// TwinCAT 3 PLC project SiftClient
// Title: Sift Client Library
// Company: Sift Stack Inc
// Author: Marc Julien
// ProjectVersion: 0.2.0.0
// Description: Sift Client library for streaming data from PLC applications into Sift.
// ProgramVersion: 3.1.4026.14
// libraries:
//   Tc2_Standard, * (Beckhoff Automation GmbH)
//   Tc2_System, * (Beckhoff Automation GmbH)
//   Tc2_TcpIp, * (Beckhoff Automation GmbH)
//   Tc2_Utilities, * (Beckhoff Automation GmbH)
//   Tc3_JsonXml, * (Beckhoff Automation GmbH)
//   TcUnit, * (www.tcunit.org)
// project tree:
//   DUTs/ E_ChannelDataType.TcDUT, ST_ChannelConfig.TcDUT, ST_EnumType.TcDUT, ST_FlowConfig.TcDUT, ST_IngestionConfig.TcDUT, T_SiftClient.TcDUT, ST_SiftError.TcDUT
//   DUTs/Private/ _ST_Timestamp.TcDUT, _ST_SiftMessage.TcDUT, _U_SiftChannelValue.TcDUT
//   GVLs/ GVL_SIFT.TcGVL, SiftClientParameters.TcGVL
//   / PlcTask.TcTTO
//   POUs/ FB_SiftClient.TcPOU
//   POUs/Private/ SAFE_MEMCPY.TcPOU, _FB_SendSiftMessage.TcPOU, _FB_BufferWriter.TcPOU, _F_CreateAuthenticateMessage.TcPOU, _F_CreateDataMessage.TcPOU, _F_CreateEndpointMessage.TcPOU, _F_CreateIngestionConfigMessage.TcPOU, _F_CreatePingMessage.TcPOU, _F_CreateRunMessage.TcPOU, _F_IsSuccessfulResponse.TcPOU, _F_SetSiftError.TcPOU
//   POUs/Services/ FB_IngestionConfigService.TcPOU, FB_IngestService.TcPOU, FB_PingService.TcPOU, FB_RunService.TcPOU
//   POUs/Services/Private/ FB_AuthenticateService.TcPOU
//   POUs/Util/ GetCurrentTime.TcPOU, SetChannelValue.TcPOU
//   Tests/ FB_BufferWriter_Test.TcPOU, FB_CreateDataMessage_Test.TcPOU, FB_CreateIngestionConfigMessage_Test.TcPOU, FB_CreatePingMessage_Test.TcPOU, FB_CreateRunMessage_Test.TcPOU, FB_SAFE_MEMCPY_Test.TcPOU, FB_SetChannelValue_Test.TcPOU, FB_SiftError_Test.TcPOU, PRG_TEST.TcPOU
//   Version/ Global_Version.TcGVL
// real-time tasks:
//   TASK PlcTask: cycle T#10ms, priority 20, ADS port 350

CONFIGURATION SiftClient
    RESOURCE PLC ON TwinCAT3
        TASK PlcTask(INTERVAL := T#10ms, PRIORITY := 20);
        PROGRAM PRG_TEST WITH PlcTask : PRG_TEST;
    END_RESOURCE
END_CONFIGURATION

// ---- DUTs/E_ChannelDataType.TcDUT
{attribute 'qualified_only'}
{attribute 'strict'}
{attribute 'to_string'}
TYPE E_ChannelDataType :
(
	Unspecified,
	Int32,
	Uint32,
	Int64,
	Uint64,
	Bool_,
	String_,
	Double,
	Float,
	Enum
);
END_TYPE

// ---- DUTs/Private/_ST_Timestamp.TcDUT
TYPE _ST_Timestamp :
STRUCT
	nSeconds : LINT;
	nNanoseconds : DINT;
END_STRUCT
END_TYPE

// ---- DUTs/Private/_ST_SiftMessage.TcDUT
TYPE _ST_SiftMessage :
STRUCT
	nType : BYTE;
	nLength : UDINT;
	aData : ARRAY[1..SiftClientParameters.MAX_PACKET_SIZE] OF BYTE;
END_STRUCT
END_TYPE

// ---- DUTs/Private/_U_SiftChannelValue.TcDUT
TYPE _U_SiftChannelValue :
UNION
	nInt32 : DINT;
	nUint32 : UDINT;
	nInt64 : LINT;
	nUint64 : ULINT;
	bBool : BOOL;
	fDouble : LREAL;
	fFloat : REAL;
	nEnum : UDINT;
	sString : STRING(255);
END_UNION
END_TYPE

// ---- DUTs/ST_ChannelConfig.TcDUT
TYPE ST_ChannelConfig :
STRUCT
	sName : STRING(255); 		   // This Channel's name. Required.
	eDataType : E_ChannelDataType; // This Channel's data type. Required.
	sDescription : STRING(255);	   // This Channel's description. Optional.
	sUnit : STRING(255);           // This Channel's units. Optional.
	// Enums for this channel. Required for Channels with the Enum data type.
	aEnumTypes : ARRAY[0..SiftClientParameters.MAX_NUM_ENUMS_PER_CHANNEL - 1] OF ST_EnumType;
	nNumEnumTypes : UDINT; // Total number of enums for this Channel.
	
	Value : _U_SiftChannelValue; // The current value of this Channel.
END_STRUCT
END_TYPE

// ---- DUTs/ST_EnumType.TcDUT
TYPE ST_EnumType :
STRUCT
	nKey : UDINT;        // Numerical key for this Enum.
	sName : STRING(255); // Name or label for this Enum.
END_STRUCT
END_TYPE

// ---- DUTs/ST_FlowConfig.TcDUT
TYPE ST_FlowConfig :
STRUCT
	sName : STRING(255); // This Flow's name.
	// The Channels in this Flow.
	aChannelConfigs : ARRAY[0..SiftClientParameters.MAX_NUM_CHANNELS_PER_FLOW - 1] OF ST_ChannelConfig;
	nNumChannelConfigs : UDINT; // Total number of channels in this Flow.
END_STRUCT
END_TYPE

// ---- DUTs/ST_IngestionConfig.TcDUT
TYPE ST_IngestionConfig :
STRUCT
	sAssetName : STRING(255); // Asset name for this Ingestion Config.
	// The Flows for this Ingestion Config.
	aFlowConfigs : ARRAY[0..SiftClientParameters.MAX_NUM_FLOWS - 1] OF ST_FlowConfig;
	nNumFlowConfigs : UDINT; // Total number of Flows in this Ingestion Config.
END_STRUCT
END_TYPE

// ---- DUTs/T_SiftClient.TcDUT
TYPE T_SiftClient :
STRUCT
	sHost : T_IPv4Addr; // Sift Proxy address.
	nPort : UINT;       // Sift Proxy port.
	
	sGrpcUri : STRING(255); // Sift gRPC URI.
	sApiKey : STRING;       // Sift API key.
	
	pJsonBuffer : POINTER TO BYTE; // Buffer used to create JSON messages.
	pJbLength : UDINT;			   // Size of pJsonBuffer.
	
   	fbCloseAll 		: FB_SocketCloseAll;
	fbConnect		: FB_SocketConnect;
	fbSend		    : FB_SocketSend;
	fbReceive     	: FB_SocketReceive;
	fbClose			: FB_SocketClose;
	
END_STRUCT
END_TYPE

// ---- DUTs/ST_SiftError.TcDUT
TYPE ST_SiftError :
STRUCT
	bError : BOOL;     // True is this is an error. 
	nErrId : UDINT;    // The ID of this error.
	sReason : STRING;  // Error message in string format.
END_STRUCT
END_TYPE

// ---- GVLs/GVL_SIFT.TcGVL
{attribute 'qualified_only'}
VAR_GLOBAL CONSTANT
	//Defaults
	SIFT_PROXY_CMD_ARGS : STRING(255) := '--stream_metrics --storage_path %s --listen_port=%d --grpc_uri=%s --api_key=%s tcp sift_proxy --little_endian --end_stream_on_error --verbose';
	SIFT_PROXY_DEFAULT_HOST : T_IPv4Addr := '127.0.0.1';
	SIFT_PROXY_DEFAULT_LISTEN_PORT : UINT := 10010;
	SIFT_PROXY_START_DELAY : TIME := T#5S;
	
	SYNC_WORD : UDINT := 16#ABCDEF00;
	HEADER_LENGTH : UDINT := 9;
	MESSAGE_TYPE_INDEX : BYTE := 4;
	MESSGE_LENGTH_INDEX : BYTE := 5;

	ENDPOINT_MESSAGE_TYPE : BYTE := 16#01;
	DATA_MESSAGE_TYPE : BYTE := 16#02;
	RESPONSE_MESSAGE_TYPE : BYTE := 16#FF;
	
	SIFT_CLIENT_DEFAULT_LOCAL_IP : T_IPv4Addr := '127.0.0.1';
	SIFT_CLIENT_DEFAULT_LOCAL_PORT : UINT := 10009;
	
	MAX_JSON_RESPONSE_SIZE : UDINT := 1024; // Max JSON response size.
		
	(* Error Codes *)
	BUFFER_CAPACITY_REACHED : UDINT := 16#5000_0000; // Buffer is at capacity.
	JSON_CAPACITY_REACHED : UDINT := 16#5000_0001; // JSON message is too large. Should increase JSON buffer size.
	NULL_JSON_POINTER : UDINT := 16#5000_0002; // The JSON buffer passed in is Null.
	INGEST_RING_BUFFER_REMOVE_ERROR : UDINT := 16#5000_0003; // Error removing data from ingest ring buffer.
	MEMCPY_ERROR : UDINT := 16#5000_0004; // Error calling MEMCPY
	BAD_PARAMETERS : UDINT := 16#5000_0005; // User has configured the parameters incorrectly.
	UNABLE_TO_PARSE_JSON : UDINT := 16#5000_0005; // Internal JSON could not be parsed.
	
	SIFT_PROXY_NO_RESPONSE : UDINT := 16#5000_1000; // No response from Sift Proxy
	SIFT_PROXY_FAILED_TO_START : UDINT := 16#5000_1001;  // Failed to start Sift Proxy
	SIFT_PROXY_INVALID_RESPONSE : UDINT := 16#5000_1002;  // Invalid response from Sift Proxy
	SIFT_PROXY_INVALID_SYNC_WORD : UDINT := 16#5000_1003;  // Invalid sync word from Sift Proxy
	SIFT_PROXY_SIFT_API_ERROR : UDINT := 16#5000_1004;  // Invalid argument to the endpoint
	
	INVALID_GRPC_URI : UDINT := 16#5000_2000;
	INVALID_API_KEY : UDINT := 16#5000_2001;
	INVALID_INGESTION_CONFIG : UDINT := 16#5000_2002;
    INVALID_LOG_DIR : UDINT := 16#5000_2003;
	
END_VAR

// ---- GVLs/SiftClientParameters.TcGVL
{attribute 'qualified_only'}
VAR_GLOBAL CONSTANT
	// The path to the `start_sift_proxy.bat` file.
	START_SIFT_PROXY_PATH : STRING := 'C:\Sift\Beckhoff\start_sift_proxy.bat';
		
	MAX_NUM_FLOWS : UDINT := 8; // Max number of Flows per Ingestion Config.
	MAX_NUM_CHANNELS_PER_FLOW : UDINT := 256; // Max number of Channels per Flow.
	MAX_NUM_ENUMS_PER_CHANNEL : UDINT := 256; // Max number of Enums per Channel.
	MAX_NUM_TAGS : UDINT := 32; // Max number of tags (for a run).
	
	// Maximum size of a single Sift packet. 
	// This should be large enough to fit all configured flows at once
	// and also large enough to fit the ingestion config request.
	MAX_PACKET_SIZE : UDINT := 8192;
	
END_VAR

// ---- Version/Global_Version.TcGVL
{attribute 'TcGenerated'}
{attribute 'no-analysis'}
{attribute 'linkalways'}
// This function has been automatically generated from the project information.
VAR_GLOBAL CONSTANT
	{attribute 'const_non_replaced'}
	stLibVersion_Sift_Client_Library : ST_LibVersion := (iMajor := 0, iMinor := 1, iBuild := 0, iRevision := 0, nFlags := 0, sVersion := '0.1.0.0');
END_VAR

// ---- Tests/PRG_TEST.TcPOU
PROGRAM PRG_TEST
VAR
	fbSetChannelValue_Test : FB_SetChannelValue_Test;
	fbSafeMemcpy_Test : FB_SAFE_MEMCPY_Test;
	fbBufferWriter_Test : FB_BufferWriter_Test;
	fbCreateIngestionConfigMessage_Test: FB_CreateIngestionConfigMessage_Test;
	fbCreatePingMessage_Test : FB_CreatePingMessage_Test;
	fbCreateRunMessage_Test : FB_CreateRunMessage_Test;
	fbSiftError_Test : FB_SiftError_Test;
	fbCreateDataMessage_Test : FB_CreateDataMessage_Test;
END_VAR

TcUnit.RUN();

END_PROGRAM

// ---- Tests/FB_SetChannelValue_Test.TcPOU
FUNCTION_BLOCK FB_SetChannelValue_Test EXTENDS TcUnit.FB_TestSuite
VAR_INPUT
END_VAR

VAR_OUTPUT
END_VAR

VAR
	stIngestionConfig : ST_IngestionConfig;
	fbIngestionConfig : FB_IngestionConfigService := (stIngestionConfig := stIngestionConfig);
	pFlowConfig : POINTER TO ST_FlowConfig;
	pChannel : POINTER TO ST_ChannelConfig;
END_VAR

Nominal();
Invalid();

METHOD Invalid : REFERENCE TO FB_Test
VAR_INPUT
	bBoolTestValue : BOOL := TRUE;
	fDoubleTestValue : LREAL := 1.2345;
	nEnumTestValue : UDINT := 10;
	fFloatTestValue : REAL := 9.8765;
	nInt32TestValue : DINT := 12345;
	sStringTestValue : STRING(255) := 'Test string value';
	nUInt32TestValue : UDINT := 4893573;
	nInt64TestValue : LINT := -12232423;
	nUInt64TestValue : ULINT := 1249864785;
END_VAR
TEST('SetChannelValue Invalid');

pFlowConfig := fbIngestionConfig.CreateFlowConfig('flow_name');

// Null
AssertFalse(SetChannelValue(pChannel := pChannel, fDoubleTestValue),
            Message := 'setting a null pointer should have failed');

// BOOL
pChannel := fbIngestionConfig.CreateChannelConfig(pFlowConfig := pFlowConfig,
                                                  sName := 'bool_channel',
                                                  E_ChannelDataType.Bool_,
                                                  sDescription := '',
                                                  sUnit := '');				  
AssertFalse(SetChannelValue(pChannel := pChannel, fDoubleTestValue),
            Message := 'setting the bool value should have failed');

// STRING
pChannel := fbIngestionConfig.CreateChannelConfig(pFlowConfig := pFlowConfig,
                                                  sName := 'string_channel',
                                                  E_ChannelDataType.String_,
                                                  sDescription := '',
                                                  sUnit := '');
AssertFalse(SetChannelValue(pChannel := pChannel, nUInt32TestValue),
            Message := 'setting the string value should have failed');

// DOUBLE
pChannel := fbIngestionConfig.CreateChannelConfig(pFlowConfig := pFlowConfig,
                                                  sName := 'double_channel',
                                                  E_ChannelDataType.Double,
                                                  sDescription := '',
                                                  sUnit := '');				  
AssertFalse(SetChannelValue(pChannel := pChannel, nEnumTestValue),
            Message := 'setting the string value should have failed');

// FLOAT
pChannel := fbIngestionConfig.CreateChannelConfig(pFlowConfig := pFlowConfig,
                                                  sName := 'float_channel',
                                                  E_ChannelDataType.Float,
                                                  sDescription := '',
                                                  sUnit := '');				  
AssertFalse(SetChannelValue(pChannel := pChannel, nInt32TestValue),
            Message := 'setting the float value should have failed');

// ENUM
pChannel := fbIngestionConfig.CreateChannelConfig(pFlowConfig := pFlowConfig,
                                                  sName := 'enum_channel',
                                                  E_ChannelDataType.Enum,
                                                  sDescription := '',
                                                  sUnit := '');				  
AssertFalse(SetChannelValue(pChannel := pChannel, fFloatTestValue),
            Message := 'setting the enum value should have failed');

// INT32
pChannel := fbIngestionConfig.CreateChannelConfig(pFlowConfig := pFlowConfig,
                                                  sName := 'int32_channel',
                                                  E_ChannelDataType.Int32,
                                                  sDescription := '',
                                                  sUnit := '');				  
AssertFalse(SetChannelValue(pChannel := pChannel, sStringTestValue),
            Message := 'setting the int32 value should have failed');

// UINT32
pChannel := fbIngestionConfig.CreateChannelConfig(pFlowConfig := pFlowConfig,
                                                  sName := 'uint32_channel',
                                                  E_ChannelDataType.Uint32,
                                                  sDescription := '',
                                                  sUnit := '');				  
AssertFalse(SetChannelValue(pChannel := pChannel, nInt64TestValue),
            Message := 'setting the uint32 value should have failed');

// INT64
pChannel := fbIngestionConfig.CreateChannelConfig(pFlowConfig := pFlowConfig,
                                                  sName := 'int64_channel',
                                                  E_ChannelDataType.Int64,
                                                  sDescription := '',
                                                  sUnit := '');				  
AssertFalse(SetChannelValue(pChannel := pChannel, nUInt64TestValue),
            Message := 'setting the int64 value should have failed');

// UINT64
pChannel := fbIngestionConfig.CreateChannelConfig(pFlowConfig := pFlowConfig,
                                                  sName := 'uint64_channel',
                                                  E_ChannelDataType.Uint64,
                                                  sDescription := '',
                                                  sUnit := '');				  
AssertFalse(SetChannelValue(pChannel := pChannel, bBoolTestValue),
            Message := 'setting the uint64 value should have failed');


TEST_FINISHED();
END_METHOD

METHOD Nominal : REFERENCE TO FB_Test
VAR_INPUT
END_VAR

VAR
	bBoolTestValue : BOOL := TRUE;
	fDoubleTestValue : LREAL := 1.2345;
	nEnumTestValue : UDINT := 10;
	fFloatTestValue : REAL := 9.8765;
	nInt32TestValue : DINT := 12345;
	sStringTestValue : STRING(255) := 'Test string value';
	nUInt32TestValue : UDINT := 4893573;
	nInt64TestValue : LINT := -12232423;
	nUInt64TestValue : ULINT := 1249864785;
END_VAR
TEST('SetChannelValue Nominal');

pFlowConfig := fbIngestionConfig.CreateFlowConfig('flow_name');

// BOOL
pChannel := fbIngestionConfig.CreateChannelConfig(pFlowConfig := pFlowConfig,
                                                  sName := 'bool_channel',
                                                  E_ChannelDataType.Bool_,
                                                  sDescription := '',
                                                  sUnit := '');				  
AssertTrue(SetChannelValue(pChannel := pChannel, bBoolTestValue),
           Message := 'the bool value was not set correctly');
AssertEquals_BOOL(Expected := bBoolTestValue, 
                  Actual := pChannel^.Value.bBool,
                  Message := 'the bool value is incorrect');

// STRING
pChannel := fbIngestionConfig.CreateChannelConfig(pFlowConfig := pFlowConfig,
                                                  sName := 'string_channel',
                                                  E_ChannelDataType.String_,
                                                  sDescription := '',
                                                  sUnit := '');
AssertTrue(SetChannelValue(pChannel := pChannel, sStringTestValue),
           Message := 'the string value was not set correctly');
AssertEquals_STRING(Expected := sStringTestValue, 
                    Actual := pChannel^.Value.sString,
                    Message := 'the string value is incorrect');

// DOUBLE
pChannel := fbIngestionConfig.CreateChannelConfig(pFlowConfig := pFlowConfig,
                                                  sName := 'double_channel',
                                                  E_ChannelDataType.Double,
                                                  sDescription := '',
                                                  sUnit := '');				  
AssertTrue(SetChannelValue(pChannel := pChannel, fDoubleTestValue),
           Message := 'the double value was not set correctly');
AssertEquals_LREAL(Expected := fDoubleTestValue, 
                   Actual := pChannel^.Value.fDouble,
                   Message := 'the double value is incorrect',
                   Delta := 0.0);

// FLOAT
pChannel := fbIngestionConfig.CreateChannelConfig(pFlowConfig := pFlowConfig,
                                                  sName := 'float_channel',
                                                  E_ChannelDataType.Float,
                                                  sDescription := '',
                                                  sUnit := '');				  
AssertTrue(SetChannelValue(pChannel := pChannel, fFloatTestValue),
           Message := 'the float value was not set correctly');
AssertEquals_REAL(Expected := fFloatTestValue, 
                  Actual := pChannel^.Value.fFloat,
                  Message := 'the float value is incorrect',
                  Delta := 0.0);

// ENUM
pChannel := fbIngestionConfig.CreateChannelConfig(pFlowConfig := pFlowConfig,
                                                  sName := 'enum_channel',
                                                  E_ChannelDataType.Enum,
                                                  sDescription := '',
                                                  sUnit := '');				  
AssertTrue(SetChannelValue(pChannel := pChannel, nEnumTestValue),
           Message := 'the enum value was not set correctly');
AssertEquals_UDINT(Expected := nEnumTestValue, 
                   Actual := pChannel^.Value.nEnum,
                   Message := 'the enum value is incorrect');

// INT32
pChannel := fbIngestionConfig.CreateChannelConfig(pFlowConfig := pFlowConfig,
                                                  sName := 'int32_channel',
                                                  E_ChannelDataType.Int32,
                                                  sDescription := '',
                                                  sUnit := '');				  
AssertTrue(SetChannelValue(pChannel := pChannel, nInt32TestValue),
           Message := 'the int32 value was not set correctly');
AssertEquals_DINT(Expected := nInt32TestValue, 
                  Actual := pChannel^.Value.nInt32,
                  Message := 'the int32 value is incorrect');

// UINT32
pChannel := fbIngestionConfig.CreateChannelConfig(pFlowConfig := pFlowConfig,
                                                  sName := 'uint32_channel',
                                                  E_ChannelDataType.Uint32,
                                                  sDescription := '',
                                                  sUnit := '');				  
AssertTrue(SetChannelValue(pChannel := pChannel, nUInt32TestValue),
           Message := 'the uint32 value was not set correctly');
AssertEquals_UDINT(Expected := nUInt32TestValue, 
                   Actual := pChannel^.Value.nUInt32,
                   Message := 'the uint32 value is incorrect');

// INT64
pChannel := fbIngestionConfig.CreateChannelConfig(pFlowConfig := pFlowConfig,
                                                  sName := 'int64_channel',
                                                  E_ChannelDataType.Int64,
                                                  sDescription := '',
                                                  sUnit := '');				  
AssertTrue(SetChannelValue(pChannel := pChannel, nInt64TestValue),
           Message := 'the int64 value was not set correctly');
AssertEquals_LINT(Expected := nInt64TestValue, 
                  Actual := pChannel^.Value.nInt64,
                  Message := 'the int64 value is incorrect');

// UINT64
pChannel := fbIngestionConfig.CreateChannelConfig(pFlowConfig := pFlowConfig,
                                                  sName := 'uint64_channel',
                                                  E_ChannelDataType.Uint64,
                                                  sDescription := '',
                                                  sUnit := '');				  
AssertTrue(SetChannelValue(pChannel := pChannel, nUInt64TestValue),
           Message := 'the uint64 value was not set correctly');
AssertEquals_ULINT(Expected := nUInt64TestValue, 
                   Actual := pChannel^.Value.nUInt64,
                   Message := 'the uint64 value is incorrect');

TEST_FINISHED();
END_METHOD

END_FUNCTION_BLOCK

// ---- POUs/Services/FB_IngestionConfigService.TcPOU
// Service for creating and sending an Ingestion Config.
// The Ingestion Config is sent on the rising edge of bExecute.
FUNCTION_BLOCK FB_IngestionConfigService
VAR_INPUT
	hSiftClient : REFERENCE TO T_SiftClient;
	sAssetName : STRING(255);
	bExecute : BOOL;
	
END_VAR
VAR_OUTPUT
	bBusy : BOOL;
	bError : BOOL;
	nErrId : UDINT;
	sId : STRING(255);
	stIngestionConfig : ST_IngestionConfig;
	stSiftError : ST_SiftError;
END_VAR
VAR
	eState : (IDLE, SEND_MESSAGE, WAIT_FOR_RESPONSE, SUCCESS, FAILURE) := IDLE;
	fbSendSiftMessage : _FB_SendSiftMessage;
	stConfigReq : _ST_SiftMessage;
	fbJson : FB_JsonDomParser;
	sResponse : STRING(GVL_SIFT.MAX_JSON_RESPONSE_SIZE);
	jsonDoc : SJsonValue;
END_VAR

stIngestionConfig.sAssetName := sAssetName;
		
CASE eState OF
	IDLE:		
		IF bExecute THEN
			eState := SEND_MESSAGE;
		END_IF
		
	SEND_MESSAGE:
		bBusy := TRUE;
		bError := FALSE;
		stSiftError := _F_CreateIngestionConfigMessage(stIngestionConfig := stIngestionConfig, 
													   stMsg := stConfigReq,
													   pJsonBuffer := hSiftClient.pJsonBuffer,
													   nLength := hSiftClient.pJbLength);
		IF stSiftError.bError THEN
			nErrId := stSiftError.nErrId;
			eState := FAILURE;
			RETURN;
		END_IF
		fbSendSiftMessage(hSiftClient := hSiftClient, stMsg := stConfigReq, bExecute := TRUE);
		eState := WAIT_FOR_RESPONSE;

	WAIT_FOR_RESPONSE:
		bBusy := TRUE;
		bError := FALSE;
		fbSendSiftMessage(bExecute := FALSE);
		
		IF fbSendSiftMessage.bBusy THEN
			RETURN;
		ELSIF fbSendSiftMessage.bError THEN
			nErrId := fbSendSiftMessage.nErrId;
			eState := FAILURE;
			RETURN;
		END_IF
		
		// Verify response.
		IF fbSendSiftMessage.stResponse.nLength > GVL_SIFT.MAX_JSON_RESPONSE_SIZE THEN
			nErrId := GVL_SIFT.JSON_CAPACITY_REACHED;
			eState := FAILURE;
			RETURN;	
		END_IF
		
		IF NOT SAFE_MEMCPY(ADR(sResponse), SIZEOF(sResponse), 
			               ADR(fbSendSiftMessage.stResponse.aData), fbSendSiftMessage.stResponse.nLength) THEN
			nErrId := GVL_SIFT.MEMCPY_ERROR;
			eState := FAILURE;
		END_IF
		
		jsonDoc := fbJson.ParseDocument(sResponse);
		IF jsonDoc = 0 THEN
			eState := FAILURE;
			nErrId := GVL_SIFT.UNABLE_TO_PARSE_JSON;
		END_IF
		
		IF _F_IsSuccessfulResponse(jsonDoc) THEN
			IF NOT fbJson.HasMember(jsonDoc, 'data') THEN
				nErrId := GVL_SIFT.SIFT_PROXY_INVALID_RESPONSE;
				eState := FAILURE;
				RETURN;
			END_IF
			
			jsonDoc := fbJson.FindMember(jsonDoc, 'data');	
			IF NOT fbJson.HasMember(jsonDoc, 'ingestionConfig') THEN
				nErrId := GVL_SIFT.SIFT_PROXY_INVALID_RESPONSE;
				eState := FAILURE;
				RETURN;
			END_IF

			jsonDoc := fbJson.FindMember(jsonDoc, 'ingestionConfig');
			IF NOT fbJson.HasMember(jsonDoc, 'ingestionConfigId') THEN
				nErrId := GVL_SIFT.SIFT_PROXY_INVALID_RESPONSE;
				eState := FAILURE;
				RETURN;
			END_IF
			
			jsonDoc := fbJson.FindMember(jsonDoc, 'ingestionConfigId');
			sId := fbJson.GetString(jsonDoc);
			
			eState := SUCCESS;
		ELSE
			IF NOT _F_SetSiftError(jsonDoc, stSiftError) THEN
				nErrId := GVL_SIFT.SIFT_PROXY_INVALID_RESPONSE;
				RETURN;
			END_IF
			nErrId := stSiftError.nErrId;
			eState := FAILURE;
		END_IF
		
	SUCCESS:
		bBusy := FALSE;
		bError := FALSE;
		eState := IDLE;
		
	FAILURE:
		bBusy := FALSE;
		bError := TRUE;
		eState := IDLE;
END_CASE

METHOD ClearIngestionConfig : BOOL
VAR_INPUT
END_VAR

VAR
	i,j : UDINT;
END_VAR
FOR i := 1 TO stIngestionConfig.nNumFlowConfigs DO
	FOR j := 1 TO stIngestionConfig.aFlowConfigs[i-1].nNumChannelConfigs DO
    	stIngestionConfig.aFlowConfigs[i-1].aChannelConfigs[j-1].sName := '';
		stIngestionConfig.aFlowConfigs[i-1].aChannelConfigs[j-1].sDescription := '';
		stIngestionConfig.aFlowConfigs[i-1].aChannelConfigs[j-1].sUnit := '';
		stIngestionConfig.aFlowConfigs[i-1].aChannelConfigs[j-1].eDataType := E_ChannelDataType.Unspecified;
		stIngestionConfig.aFlowConfigs[i-1].aChannelConfigs[j-1].nNumEnumTypes := 0;
	END_FOR
	stIngestionConfig.aFlowConfigs[i-1].nNumChannelConfigs := 0;
	stIngestionConfig.aFlowConfigs[i-1].sName := '';
END_FOR
stIngestionConfig.sAssetName := '';
stIngestionConfig.nNumFlowConfigs := 0;
END_METHOD

METHOD CreateChannelConfig : POINTER TO ST_ChannelConfig
VAR_INPUT
	pFlowConfig : POINTER TO ST_FlowConfig;
	sName : STRING(255);
	eDataType : E_ChannelDataType;
	sDescription : STRING(255);
	sUnit : STRING(255);
END_VAR
VAR 
	pChannelConfig : POINTER TO ST_ChannelConfig;
END_VAR
IF pFlowConfig = 0 THEN
	CreateChannelConfig := 0;
	RETURN;
END_IF

IF pFlowConfig^.nNumChannelConfigs >= SiftClientParameters.MAX_NUM_CHANNELS_PER_FLOW THEN
	CreateChannelConfig := 0;
	RETURN;
END_IF

pChannelConfig := ADR(pFlowConfig^.aChannelConfigs[pFlowConfig^.nNumChannelConfigs]);
pChannelConfig^.sName := sName;
pChannelConfig^.eDataType := eDataType;
pChannelConfig^.sDescription := sDescription;
pChannelConfig^.sUnit := sUnit;

pFlowConfig^.nNumChannelConfigs := pFlowConfig^.nNumChannelConfigs + 1;
CreateChannelConfig := pChannelConfig;
END_METHOD

METHOD CreateFlowConfig : POINTER TO ST_FlowConfig
VAR_INPUT
	sName : STRING(255);
END_VAR
IF stIngestionConfig.nNumFlowConfigs >= SiftClientParameters.MAX_NUM_FLOWS THEN
	CreateFlowConfig := 0;
	RETURN;
END_IF

stIngestionConfig.aFlowConfigs[stIngestionConfig.nNumFlowConfigs].sName := sName;
CreateFlowConfig := ADR(stIngestionConfig.aFlowConfigs[stIngestionConfig.nNumFlowConfigs]);

stIngestionConfig.nNumFlowConfigs := stIngestionConfig.nNumFlowConfigs + 1;
END_METHOD

METHOD InitEnumTypes : BOOL
VAR_INPUT
	pChannelConfig : POINTER TO ST_ChannelConfig;
	aEnumTypes : REFERENCE TO ARRAY[0..SiftClientParameters.MAX_NUM_ENUMS_PER_CHANNEL - 1] OF ST_EnumType;
END_VAR

VAR 
	i : UDINT;
END_VAR
IF pChannelConfig = 0 THEN
	InitEnumTypes := FALSE;
	RETURN;
END_IF

IF pChannelConfig^.eDataType <> E_ChannelDataType.Enum THEN
	InitEnumTypes := FALSE;
	RETURN;
END_IF


FOR i := 1 TO SiftClientParameters.MAX_NUM_ENUMS_PER_CHANNEL DO
	IF aEnumTypes[i-1].sName = '' THEN
		CONTINUE;
	END_IF
	
	pChannelConfig^.aEnumTypes[i-1] := aEnumTypes[i-1];
	pChannelConfig^.nNumEnumTypes := pChannelConfig^.nNumEnumTypes + 1;
END_FOR

InitEnumTypes := TRUE;
END_METHOD

// Resets the Ingestion Config service.
METHOD PUBLIC Reset : BOOL
VAR_INPUT
END_VAR
Reset := ClearIngestionConfig();
END_METHOD

METHOD PUBLIC Validate : BOOL
VAR_INPUT
END_VAR
VAR
	nSizeInBytes : UDINT;
	i : UDINT;
	j : UDINT;
	tmpChannelConfig : REFERENCE TO ST_ChannelConfig;
END_VAR
FOR i := 1 TO stIngestionConfig.nNumFlowConfigs DO
	FOR j := 1 TO stIngestionConfig.aFlowConfigs[i-1].nNumChannelConfigs DO
		tmpChannelConfig REF= stIngestionConfig.aFlowConfigs[i-1].aChannelConfigs[j-1];

		CASE tmpChannelConfig.eDataType OF
			E_ChannelDataType.Bool_:
				nSizeInBytes := nSizeInBytes + 1;
			
			E_ChannelDataType.Double:
				nSizeInBytes := nSizeInBytes + 8;
			
			E_ChannelDataType.Enum:
				nSizeInBytes := nSizeInBytes + 4;
			
			E_ChannelDataType.Float:
				nSizeInBytes := nSizeInBytes + 4;
			
			E_ChannelDataType.Int32:
				nSizeInBytes := nSizeInBytes + 4;
			
			E_ChannelDataType.Int64:
				nSizeInBytes := nSizeInBytes + 8;
			
			E_ChannelDataType.String_:
				nSizeInBytes := nSizeInBytes + 255;
			
			E_ChannelDataType.Uint32:
				nSizeInBytes := nSizeInBytes + 4;

			E_ChannelDataType.Uint64:
				nSizeInBytes := nSizeInBytes + 8;
		END_CASE
		
		IF tmpChannelConfig.eDataType = E_ChannelDataType.Unspecified THEN
			Validate := FALSE;
			RETURN;
		END_IF
	END_FOR
END_FOR

Validate := nSizeInBytes < SiftClientParameters.MAX_PACKET_SIZE;
END_METHOD

END_FUNCTION_BLOCK

// ---- POUs/Private/_FB_SendSiftMessage.TcPOU
// Sends a message to Sift Proxy using the Sift Proxy Protocol and waits for a response.
FUNCTION_BLOCK _FB_SendSiftMessage
VAR_INPUT
	hSiftClient : REFERENCE TO T_SiftClient;
	stMsg : REFERENCE TO _ST_SiftMessage;
	bExecute : BOOL;
	bWaitForReply : BOOL := TRUE;
	tReplyTimeout : TIME := T#10S; // Default 10s timeout. In practice we've seen local repsonses take up to about 1s.
END_VAR
VAR_OUTPUT
	bBusy : BOOL;
	bError : BOOL;
	stResponse : _ST_SiftMessage;
	nErrId : UDINT;
END_VAR

VAR
	eState : (IDLE, SEND_MESSAGE, SEND_MESSAGE_WAIT, RECEIVE_REPLY_START_TIMER, RECEIVE_REPLY, RECEIVE_REPLY_WAIT, SUCCESS, FAILURE):= IDLE;
	aRawBuf : ARRAY[1..SiftClientParameters.MAX_PACKET_SIZE] OF BYTE; // For the BufferWriter. Used for sending/receiving.
	fbWriter : _FB_BufferWriter := (pRawBuf := ADR(aRawBuf), nSize := SIZEOF(aRawBuf));	
	aRecvBuf : ARRAY[1..SiftClientParameters.MAX_PACKET_SIZE] OF BYTE; // Used for immediate recv calls.
	responseTimer : TON; // Timer for how longer to wait for a response from sift_proxy.
	nBytesRead : UDINT; // Current offset into the recv message.
	nRecvSyncWord : UDINT;	
	nRecvCount : UDINT;
END_VAR

CASE eState OF
	IDLE:
		IF bExecute THEN
			eState := SEND_MESSAGE;
		END_IF
		
	SEND_MESSAGE:
		bBusy := TRUE;
		bError := FALSE;
		
		// Always reset the writer before using it.
		fbWriter.SetOffset(0);
		
		// Verify MAX_PACKET_SIZE is a reasonable number
		IF SiftClientParameters.MAX_PACKET_SIZE <= GVL_SIFT.HEADER_LENGTH THEN
			nErrId := GVL_SIFT.BAD_PARAMETERS;
			eState := FAILURE;
			RETURN;
		END_IF
		
		// Sync word
		IF NOT fbWriter.Write(ADR(GVL_SIFT.SYNC_WORD), 4) THEN
			nErrId := GVL_SIFT.MEMCPY_ERROR;
			eState := FAILURE;
			RETURN;
		END_IF
		
		// Message type		
		IF NOT fbWriter.Write(ADR(stMsg.nType), 1) THEN
			nErrId := GVL_SIFT.MEMCPY_ERROR;
			eState := FAILURE;
			RETURN;
		END_IF
		
		// Message length
		IF NOT fbWriter.Write(ADR(stMsg.nLength), 4) THEN
			nErrId := GVL_SIFT.MEMCPY_ERROR;
			eState := FAILURE;
			RETURN;
		END_IF
			
		// Data.
		IF NOT fbWriter.Write(ADR(stMsg.aData), stMsg.nLength) THEN
			nErrId := GVL_SIFT.MEMCPY_ERROR;
			eState := FAILURE;
			RETURN;
		END_IF
		
		hSiftClient.fbSend(
			hSocket := hSiftClient.fbConnect.hSocket, 
			pSrc := ADR(aRawBuf),
			cbLen := stMsg.nLength + GVL_SIFT.HEADER_LENGTH,
			bExecute := TRUE,
		);
	
		eState := SEND_MESSAGE_WAIT;

	SEND_MESSAGE_WAIT:
		bBusy := TRUE;
		bError := FALSE;
		hSiftClient.fbSend(bExecute := FALSE);
		
		IF hSiftClient.fbSend.bBusy THEN
			RETURN;
		ELSIF hSiftClient.fbSend.bError THEN
			nErrId := hSiftClient.fbSend.nErrId;
			eState := FAILURE;
			RETURN;
		END_IF
		
		IF bWaitForReply THEN
			eState := RECEIVE_REPLY_START_TIMER;
		ELSE
			eState := SUCCESS;
		END_IF
	
	RECEIVE_REPLY_START_TIMER:
		bBusy := TRUE;
		bError := FALSE;
		responseTimer(IN:=FALSE);
		responseTimer(IN:=TRUE, PT:=tReplyTimeout);
		eState := RECEIVE_REPLY;
		nBytesRead := 0;
		
	RECEIVE_REPLY:
		bBusy := TRUE;
		bError := FALSE;

		hSiftClient.fbReceive(
			hSocket := hSiftClient.fbConnect.hSocket,
			cbLen := SiftClientParameters.MAX_PACKET_SIZE,
			pDest := ADR(aRecvBuf),
			bExecute := TRUE,
		);
		eState := RECEIVE_REPLY_WAIT;
		
	RECEIVE_REPLY_WAIT:
		bBusy := TRUE;
		bError := FALSE;
		hSiftClient.fbReceive(bExecute := FALSE);
		responseTimer();
				
		IF hSiftClient.fbReceive.bBusy THEN
			RETURN;
		ELSIF hSiftClient.fbReceive.bError THEN
			IF responseTimer.Q THEN
				nErrId := hSiftClient.fbReceive.nErrId;
				eState := FAILURE;
			ELSE
				eState := RECEIVE_REPLY;
			END_IF
			RETURN;
		END_IF
		
		IF hSiftClient.fbReceive.nRecBytes = 0 THEN
			IF responseTimer.Q THEN
				eState := FAILURE;
				nErrId := GVL_SIFT.SIFT_PROXY_NO_RESPONSE;
			ELSE	
				eState := RECEIVE_REPLY;
			END_IF		
			RETURN;
		END_IF
		
		// Always reset the writer before using it.
		fbWriter.SetOffset(0);
			
		IF NOT fbWriter.Write(ADR(aRecvBuf), hSiftClient.fbReceive.nRecBytes) THEN
			nErrId := GVL_SIFT.MEMCPY_ERROR;
			eState := FAILURE;
			RETURN;
		END_IF
		
		// If we have a complete header.
		IF fbWriter.nCurOffset >= GVL_SIFT.HEADER_LENGTH THEN
			IF NOT SAFE_MEMCPY(ADR(nRecvSyncWord), SIZEOF(nRecvSyncWord), ADR(aRawBuf), 4) THEN
				nErrId := GVL_SIFT.MEMCPY_ERROR;
				eState := FAILURE;
				RETURN;
			END_IF
			IF nRecvSyncWord <> GVL_SIFT.SYNC_WORD THEN
				eState := FAILURE;
				nErrId := GVL_SIFT.SIFT_PROXY_INVALID_SYNC_WORD;;
				RETURN;
			END_IF
			
			stResponse.nType := aRawBuf[GVL_SIFT.MESSAGE_TYPE_INDEX+1];
			IF stResponse.nType <> GVL_SIFT.RESPONSE_MESSAGE_TYPE THEN
				eState := FAILURE;
				nErrId := GVL_SIFT.SIFT_PROXY_INVALID_RESPONSE;;
				RETURN;
			END_IF	
			
			IF NOT SAFE_MEMCPY(ADR(stResponse.nLength), SIZEOF(stResponse.nLength), ADR(aRawBuf[GVL_SIFT.MESSGE_LENGTH_INDEX+1]), 4) THEN
				nErrId := GVL_SIFT.MEMCPY_ERROR;
				eState := FAILURE;
				RETURN;
			END_IF

			// Verify that the size of this message isn't larger than our buffer.
			IF stResponse.nLength > SIZEOF(stResponse.aData) THEN
				eState := FAILURE;
				nErrId := GVL_SIFT.BUFFER_CAPACITY_REACHED;
				RETURN;
			END_IF
			
			// Check if we have the whole packet
			IF fbWriter.nCurOffset >= GVL_SIFT.HEADER_LENGTH + stResponse.nLength THEN
				IF NOT SAFE_MEMCPY(ADR(stResponse.aData), SIZEOF(stResponse.aData),
								   ADR(aRawBuf[GVL_SIFT.HEADER_LENGTH+1]), stResponse.nLength) THEN
					nErrId := GVL_SIFT.MEMCPY_ERROR;
					eState := FAILURE;
					RETURN;
				END_IF
				
			ELSE // Incomplete packet.
				eState := RECEIVE_REPLY;
				RETURN;
			END_IF

		ELSE // Incomplete header.
			eState := RECEIVE_REPLY;
			RETURN;
		END_IF
		
		eState := SUCCESS;
		
	SUCCESS:
		bBusy := FALSE;
		bError := FALSE;
		eState := IDLE;
		
	FAILURE:
		bBusy := FALSE;
		bError := TRUE;
		eState := IDLE;
END_CASE

END_FUNCTION_BLOCK

// ---- POUs/Private/_FB_BufferWriter.TcPOU
// Helper for writing bytes to an array buffer.
FUNCTION_BLOCK _FB_BufferWriter
VAR_INPUT
	pRawBuf : POINTER TO BYTE; 
	nSize : UDINT;
END_VAR

VAR_OUTPUT
	nCurOffset : UDINT;
END_VAR

VAR
END_VAR

METHOD SetOffset : BOOL
VAR_INPUT
	nOffset : UDINT;
END_VAR
IF nOffset >= nSize THEN
	SetOffset := FALSE;
ELSE
	nCurOffset := nOffset;	
	SetOffset := TRUE;
END_IF
END_METHOD

METHOD Write : BOOL
VAR_INPUT
	pSrc : POINTER TO BYTE;
	nBytes : UDINT;
END_VAR
IF nCurOffset + nBytes > nSize THEN
	Write := FALSE;
ELSE
	Write := SAFE_MEMCPY(ADR(pRawBuf[nCurOffset]), nSize, pSrc, nBytes);
	nCurOffset := nCurOffset + nBytes;	
END_IF
END_METHOD

METHOD WriteAt : BOOL
VAR_INPUT
	nIndex : UDINT;
	pSrc : POINTER TO BYTE;
	nBytes : UDINT;
END_VAR
WriteAt := SAFE_MEMCPY(ADR(pRawBuf[nIndex]), nSize-nIndex, pSrc, nBytes);
END_METHOD

METHOD WriteByte : BOOL
VAR_INPUT
	nByte : BYTE;
END_VAR
IF nCurOffset < nSize THEN
	pRawBuf[nCurOffset] := nByte;
	nCurOffset := nCurOffset + 1;
	WriteByte := TRUE;
ELSE
	WriteByte := FALSE;
END_IF
END_METHOD

END_FUNCTION_BLOCK

// ---- POUs/Private/SAFE_MEMCPY.TcPOU
// Safe version of MEMCPY. Checks NULL pointers and bounds before copying.
FUNCTION SAFE_MEMCPY : BOOL

VAR_INPUT
	pDst : POINTER TO BYTE;
	nDstLen : UDINT;
	pSrc : POINTER TO BYTE;
	nSrcLen : UDINT;
END_VAR

VAR
	nMcErr : UDINT;
END_VAR

IF pDst = 0 OR pSrc = 0 THEN
	SAFE_MEMCPY := FALSE;
	RETURN;
END_IF

IF nDstLen < nSrcLen THEN
	SAFE_MEMCPY := FALSE;
	RETURN;
END_IF

nMcErr := MEMCPY(pDst, pSrc, nSrcLen);
IF nMcErr = 0 THEN
	SAFE_MEMCPY := FALSE;
END_IF

SAFE_MEMCPY := TRUE;

END_FUNCTION

// ---- POUs/Private/_F_CreateIngestionConfigMessage.TcPOU
// Creates a Sift Proxy Protocol "create_ingestion_config" Endpoint Message.
FUNCTION _F_CreateIngestionConfigMessage 

VAR_INPUT
	stIngestionConfig : REFERENCE TO ST_IngestionConfig;
	stMsg : REFERENCE TO _ST_SiftMessage;
	pJsonBuffer : POINTER TO BYTE;
	nLength : UDINT;
END_VAR

VAR
	fbJson : FB_JsonSaxWriter;
	i : UDINT;
	j : UDINT;
	k : UDINT;
	tmpChannelConfig : REFERENCE TO ST_ChannelConfig;
	tmpEnumType : REFERENCE TO ST_EnumType;
	pJsonString : POINTER TO STRING;
	nBytes : UDINT;
END_VAR

VAR_OUTPUT
	stErr : ST_SiftError;
END_VAR

IF pJsonBuffer = 0 THEN
	stErr.bError := TRUE;
	stErr.nErrId := GVL_SIFT.NULL_JSON_POINTER;
	stErr.sReason := 'The JSON buffer is null';
	RETURN;
END_IF

fbJson.StartObject();

fbJson.AddKey('assetName');
fbJson.AddString(stIngestionConfig.sAssetName);

fbJson.AddKey('flows');
fbJson.StartArray();
FOR i := 1 TO stIngestionConfig.nNumFlowConfigs DO
	fbJson.StartObject();

	fbJson.AddKey('name');
	fbJson.AddString(stIngestionConfig.aFlowConfigs[i-1].sName);

	fbJson.AddKey('channels');
	fbJson.StartArray();
	FOR j := 1 TO stIngestionConfig.aFlowConfigs[i-1].nNumChannelConfigs DO
		fbJson.StartObject();
		tmpChannelConfig REF= stIngestionConfig.aFlowConfigs[i-1].aChannelConfigs[j-1];

		fbJson.AddKey('name');
		fbJson.AddString(tmpChannelConfig.sName);

		IF tmpChannelConfig.sUnit <> '' THEN
			fbJson.AddKey('unit');
			fbJson.AddString(tmpChannelConfig.sUnit);
		END_IF
		
		IF tmpChannelConfig.sDescription <> '' THEN
			fbJson.AddKey('description');
			fbJson.AddString(tmpChannelConfig.sDescription);
		END_IF
	
		fbJson.AddKey('dataType');
		CASE tmpChannelConfig.eDataType OF
			E_ChannelDataType.Bool_:
				fbJson.AddString('CHANNEL_DATA_TYPE_BOOL');
			
			E_ChannelDataType.Double:
				fbJson.AddString('CHANNEL_DATA_TYPE_DOUBLE');
			
			E_ChannelDataType.Enum:
				fbJson.AddString('CHANNEL_DATA_TYPE_ENUM');
			
			E_ChannelDataType.Float:
				fbJson.AddString('CHANNEL_DATA_TYPE_FLOAT');
			
			E_ChannelDataType.Int32:
				fbJson.AddString('CHANNEL_DATA_TYPE_INT_32');
			
			E_ChannelDataType.Int64:
				fbJson.AddString('CHANNEL_DATA_TYPE_INT_64');
			
			E_ChannelDataType.String_:
				fbJson.AddString('CHANNEL_DATA_TYPE_STRING');
			
			E_ChannelDataType.Uint32:
				fbJson.AddString('CHANNEL_DATA_TYPE_UINT_32');

			E_ChannelDataType.Uint64:
				fbJson.AddString('CHANNEL_DATA_TYPE_UINT_64');
		END_CASE
		
		fbJson.AddKey('enumTypes');
		fbJson.StartArray();
		FOR k := 1 TO tmpChannelConfig.nNumEnumTypes DO
			tmpEnumType REF= tmpChannelConfig.aEnumTypes[k-1];
			fbJson.StartObject();
			
			fbJson.AddKey('name');
			fbJson.AddString(tmpEnumType.sName);
			
			fbJson.AddKey('key');
			fbJson.AddUdint(tmpEnumType.nKey);
			
			fbJson.EndObject();
		END_FOR
		fbJson.EndArray();
		
		fbJson.EndObject();
	END_FOR
	fbJson.EndArray();
		
	fbJson.EndObject();
END_FOR
fbJson.EndArray();

fbJson.EndObject();

pJsonString := pJsonBuffer;
nBytes := fbJson.CopyDocument(pJsonString^, nLength);
IF nBytes = 0 THEN
	stErr.nErrId := GVL_SIFT.JSON_CAPACITY_REACHED;
	stErr.bError := TRUE;
	stErr.sReason := CONCAT(
		CONCAT('JSON msg too large: ', UDINT_TO_STRING(fbJson.GetDocumentLength())),
		' endpoint=create_ingestion_config',
	);
	RETURN;
END_IF

stErr := _F_CreateEndpointMessage(sEndpoint:='create_ingestion_config', 
                                  pData:=pJsonString, 
                                  nLength:=nBytes-1,
                                  nBufferLength := nLength, 
                                  stMsg:=stMsg);

END_FUNCTION

// ---- POUs/Private/_F_CreateEndpointMessage.TcPOU
// Creates a Sift Proxy Protocol Endpoint Message.
FUNCTION _F_CreateEndpointMessage 
VAR_INPUT
	sEndpoint : STRING; 
	pData : POINTER TO STRING;
	nLength : UDINT;
	nBufferLength : UDINT;
	stMsg : REFERENCE TO _ST_SiftMessage;
END_VAR

VAR
	fbJson : FB_JsonSaxWriter;
	nBytes : UDINT;
END_VAR

VAR_OUTPUT
	stErr : ST_SiftError;
END_VAR

IF nLength > nBufferLength THEN
	stErr.bError := TRUE;
	stErr.nErrId := GVL_SIFT.JSON_CAPACITY_REACHED;
	stErr.sReason := CONCAT(
		CONCAT('JSON msg too large: ', UDINT_TO_STRING(nLength)),
		CONCAT(' endpoint= ', sEndpoint),
	);
END_IF

fbJson.StartObject();
fbJson.AddKey('endpoint');
fbJson.AddString(sEndpoint);
fbJson.AddKey('data');
fbJson.AddRawObject(pData^);
fbJson.EndObject();

nBytes := fbJson.CopyDocument(pData^, nBufferLength);

IF nBytes = 0 THEN
	stErr.bError := TRUE;
	stErr.nErrId := GVL_SIFT.JSON_CAPACITY_REACHED;
	RETURN;
END_IF

// Omit null delimeter.
nBytes := nBytes - 1;

IF nBytes > SIZEOF(stMsg.aData) THEN
	stErr.bError := TRUE;
	stErr.nErrId := GVL_SIFT.BUFFER_CAPACITY_REACHED;
	stErr.sReason := CONCAT(
		CONCAT('Increase MAX_PACKET_SIZE. Message is too large: ', UDINT_TO_STRING(nBytes)),
		CONCAT(' endpoint= ', sEndpoint),
	);
	RETURN;
END_IF

IF NOT SAFE_MEMCPY(ADR(stMsg.aData), SIZEOF(stMsg.aData), 
				   pData, nBytes) THEN
	stErr.bError := TRUE;
	stErr.nErrId := GVL_SIFT.MEMCPY_ERROR;
	stErr.sReason := 'MEMCPY failed in CreateEndpointMessage';
	RETURN;
END_IF

stMsg.nType := GVL_SIFT.ENDPOINT_MESSAGE_TYPE;
stMsg.nLength := nBytes;

END_FUNCTION

// ---- POUs/Private/_F_IsSuccessfulResponse.TcPOU
// Returns True if the response indicates success.
FUNCTION _F_IsSuccessfulResponse : BOOL
VAR_INPUT
	jsonDoc : SJsonValue;
END_VAR
VAR
	fbJson : FB_JsonDomParser;
	jsonProp : SJsonValue;
END_VAR

IF NOT fbJson.HasMember(jsonDoc, 'status') THEN
	_F_IsSuccessfulResponse := FALSE;
	RETURN;
END_IF

jsonProp := fbJson.FindMember(jsonDoc, 'status');
_F_IsSuccessfulResponse := fbJson.GetBool(jsonProp);

END_FUNCTION

// ---- POUs/Private/_F_SetSiftError.TcPOU
// Set stSiftError to the contents of the JSON.
FUNCTION _F_SetSiftError : BOOL
VAR_INPUT
	jsonDoc : SJsonValue;
	stSiftError : REFERENCE TO ST_SiftError; 
END_VAR
VAR
	fbJson : FB_JsonDomParser;
	jsonProp : SJsonValue;
END_VAR

IF NOT fbJson.HasMember(jsonDoc, 'status') THEN
	_F_SetSiftError := FALSE;
	RETURN;
END_IF

jsonProp := fbJson.FindMember(jsonDoc, 'status');
stSiftError.bError := NOT fbJson.GetBool(jsonProp);
	
IF NOT fbJson.HasMember(jsonDoc, 'data') THEN
	_F_SetSiftError := FALSE;
	RETURN;
END_IF

jsonProp := fbJson.FindMember(jsonDoc, 'data');
IF NOT fbJson.HasMember(jsonProp, 'reason') THEN
	_F_SetSiftError := FALSE;
	RETURN;
END_IF

jsonProp := fbJson.FindMember(jsonProp, 'reason');
stSiftError.sReason := fbJson.GetString(jsonProp);

stSiftError.nErrId := GVL_SIFT.SIFT_PROXY_SIFT_API_ERROR;
stSiftError.bError := TRUE;

_F_SetSiftError := TRUE;

END_FUNCTION

// ---- POUs/Util/SetChannelValue.TcPOU
// Update the value of a Sift Channel. Should be called before FB_Ingest.WriteData() to update
// the values before they are written to the Flow.
FUNCTION SetChannelValue : BOOL
VAR_INPUT
	pChannel : POINTER TO ST_ChannelConfig;
	anyValue : ANY;
END_VAR
VAR
	stChannel : REFERENCE TO ST_ChannelConfig;
	pAnyBool : POINTER TO BOOL;
	pAnyLReal : POINTER TO LREAL;
	pAnyEnum : POINTER TO UDINT;
	pAnyReal : POINTER TO REAL;
	pAnyDInt : POINTER TO DINT;
	pAnyLInt : POINTER TO LINT;
	pAnyUDInt : POINTER TO DINT;
	pAnyULInt : POINTER TO LINT;
	pAnyString : POINTER TO STRING(255);
	bOk : BOOL;
END_VAR

IF pChannel = 0 THEN
	bOk := FALSE;
	RETURN;
END_IF

stChannel REF= pChannel^;

CASE stChannel.eDataType OF
	E_ChannelDataType.Bool_:
		IF anyValue.TypeClass = __SYSTEM.TYPE_CLASS.TYPE_BOOL THEN
			pAnyBool := anyValue.pValue;
			stChannel.Value.bBool := pAnyBool^;
			bOk := TRUE;
		ELSE
			bOk := FALSE;
		END_IF

	E_ChannelDataType.Double:
		IF anyValue.TypeClass = __SYSTEM.TYPE_CLASS.TYPE_LREAL THEN
			pAnyLReal := anyValue.pValue;
			stChannel.Value.fDouble := pAnyLReal^;
			bOk := TRUE;
		ELSE
			bOk := FALSE;
		END_IF
		
	E_ChannelDataType.Enum:
		IF anyValue.TypeClass = __SYSTEM.TYPE_CLASS.TYPE_UDINT THEN
			pAnyEnum := anyValue.pValue;
			stChannel.Value.nEnum := pAnyEnum^;
			bOk := TRUE;
		ELSE
			bOk := FALSE;
		END_IF
		
	E_ChannelDataType.Float:
		IF anyValue.TypeClass = __SYSTEM.TYPE_CLASS.TYPE_REAL THEN
			pAnyReal := anyValue.pValue;
			stChannel.Value.fFloat := pAnyReal^;
			bOk := TRUE;
		ELSE
			bOk := FALSE;
		END_IF
		
	E_ChannelDataType.Int32:
		IF anyValue.TypeClass = __SYSTEM.TYPE_CLASS.TYPE_DINT THEN
			pAnyDInt := anyValue.pValue;
			stChannel.Value.nInt32 := pAnyDInt^;
			bOk := TRUE;
		ELSE
			bOk := FALSE;
		END_IF
		
	E_ChannelDataType.Int64:
		IF anyValue.TypeClass = __SYSTEM.TYPE_CLASS.TYPE_LINT THEN
			pAnyLInt := anyValue.pValue;
			stChannel.Value.nInt64 := pAnyLInt^;
			bOk := TRUE;
		ELSE
			bOk := FALSE;
		END_IF
		
	E_ChannelDataType.UInt32:
		IF anyValue.TypeClass = __SYSTEM.TYPE_CLASS.TYPE_UDINT THEN
			pAnyUDInt := anyValue.pValue;
			stChannel.Value.nInt32 := pAnyUDInt^;
			bOk := TRUE;
		ELSE
			bOk := FALSE;
		END_IF
		
	E_ChannelDataType.UInt64:
		IF anyValue.TypeClass = __SYSTEM.TYPE_CLASS.TYPE_ULINT THEN
			pAnyULInt := anyValue.pValue;
			stChannel.Value.nInt64 := pAnyULInt^;
			bOk := TRUE;
		ELSE
			bOk := FALSE;
		END_IF
		
	E_ChannelDataType.String_:
		IF anyValue.TypeClass = __SYSTEM.TYPE_CLASS.TYPE_STRING THEN
			pAnyString := anyValue.pValue;
			stChannel.Value.sString := pAnyString^;
			bOk := TRUE;
		ELSE
			bOk := FALSE;
		END_IF
END_CASE

SetChannelValue := bOk;

END_FUNCTION

// ---- Tests/FB_SAFE_MEMCPY_Test.TcPOU
FUNCTION_BLOCK FB_SAFE_MEMCPY_Test EXTENDS TcUnit.FB_TestSuite
VAR_INPUT
END_VAR

VAR_OUTPUT
END_VAR

VAR
END_VAR

Nominal();
Invalid();

METHOD Invalid : REFERENCE TO FB_Test
VAR_INPUT
END_VAR
VAR
	pSrc : ARRAY[1..10] OF BYTE;
	pDst : ARRAY[1..10] OF BYTE;
	i : BYTE;
END_VAR
TEST('SAFE_MEMCPY Invalid');

AssertFalse(SAFE_MEMCPY(ADR(pSrc), 5, ADR(pDst), 10), Message := 'SAFE_MEMCPY should have failed with small dst buffer');
AssertFalse(SAFE_MEMCPY(0, 5, ADR(pDst), 10), Message := 'SAFE_MEMCPY should have failed with null dst');
AssertFalse(SAFE_MEMCPY(ADR(pSrc), 5, 0, 10), Message := 'SAFE_MEMCPY should have failed with null src');

TEST_FINISHED();
END_METHOD

METHOD Nominal : REFERENCE TO FB_Test
VAR_INPUT
END_VAR
VAR
	pSrc : ARRAY[1..10] OF BYTE;
	pDst : ARRAY[1..10] OF BYTE;
	i : BYTE;
END_VAR
TEST('SAFE_MEMCPY Nominal');

FOR i := 1 TO 10 DO
	pSrc[i] := i * 10;
END_FOR

// Test nominal write
AssertTrue(SAFE_MEMCPY(ADR(pSrc), 10, ADR(pDst), 10), Message := 'SAFE_MEMCPY failed');
AssertArrayEquals_BYTE(Expecteds := pSrc, Actuals := pDst, 'pSrc != pDst');

// Test 0 write
AssertTrue(SAFE_MEMCPY(ADR(pSrc), 10, ADR(pDst), 0), Message := 'SAFE_MEMCPY failed writing 0 bytes');
TEST_FINISHED();
END_METHOD

END_FUNCTION_BLOCK

// ---- Tests/FB_BufferWriter_Test.TcPOU
FUNCTION_BLOCK FB_BufferWriter_Test EXTENDS TcUnit.FB_TestSuite
VAR_INPUT
END_VAR
VAR_OUTPUT
END_VAR
VAR
	aRawBuf : ARRAY[1..10] OF BYTE;
END_VAR

NominalAndInvalid();

METHOD NominalAndInvalid : REFERENCE TO FB_Test
VAR_INPUT
END_VAR

VAR
	fbWriter : _FB_BufferWriter := (pRawBuf := ADR(aRawBuf), nSize := SIZEOF(aRawBuf));
	nData : UDINT;
	// Data is written in little-endian
	aExpected1 : ARRAY[1..10] OF BYTE := [16#AA, 16#EF, 16#CD, 16#AB, 16#DD, 16#CC, 16#AB, 16#FF, 16#AA, 16#AA];
	aExpected2 : ARRAY[1..10] OF BYTE := [16#AA, 16#EF, 16#CD, 16#AB, 16#DD, 16#04, 16#03, 16#02, 16#01, 16#AA];
END_VAR
TEST('BufferWriter Nominal and Invalid');

nData := 16#ABCDEFAA;
AssertTrue(fbWriter.Write(ADR(nData), 4), Message := 'Write 1 failed');

nData := 16#FFABCCDD;
AssertTrue(fbWriter.Write(ADR(nData), 4), Message := 'Write 2 failed');

nData := 16#AAAA;
AssertTrue(fbWriter.Write(ADR(nData), 2), Message := 'Write 3 failed');

nData := 16#ABCD;
AssertFalse(fbWriter.Write(ADR(nData), 2), Message := 'buffer full, Write should have failed');

AssertArrayEquals_BYTE(Expecteds := aExpected1, Actuals := aRawBuf, Message := 'array values dont match');
AssertEquals_UDINT(Expected := 10, Actual := fbWriter.nCurOffset, Message := 'incorrect BufferedWriter offset');

nData := 16#01020304;
AssertTrue(fbWriter.WriteAt(5, ADR(nData), 4), Message := 'BufferWriter::WriteAt 1 failed');
AssertArrayEquals_BYTE(Expecteds := aExpected2, Actuals := aRawBuf, Message := 'WriteAt did not correctly write data');
AssertEquals_UDINT(Expected := 10, Actual := fbWriter.nCurOffset, Message := 'BufferedWriter offset should not change with WriteAt');

fbWriter.SetOffset(3);
AssertTrue(fbWriter.WriteByte(16#05), Message := 'BufferWriter::WriteByte 1 failed');
AssertEquals_BYTE(Expected := 16#05, Actual := aRawBuf[4], Message := 'WriteByte did not correctly write data');
AssertEquals_UDINT(Expected := 4, Actual := fbWriter.nCurOffset, Message := 'Incorrect BufferedWriter offset after WriteByte');

TEST_FINISHED();
END_METHOD

END_FUNCTION_BLOCK

// ---- Tests/FB_CreateIngestionConfigMessage_Test.TcPOU
FUNCTION_BLOCK FB_CreateIngestionConfigMessage_Test EXTENDS TcUnit.FB_TestSuite
VAR_INPUT
END_VAR

VAR_OUTPUT
END_VAR

VAR
	fbIngestionConfig : FB_IngestionConfigService;
	aEnums : ARRAY[1..SiftClientParameters.MAX_NUM_ENUMS_PER_CHANNEL] OF ST_EnumType := [
		(nKey:=0, sName:='enum1'),
		(nKey:=1, sName:='enum2'),
		(nKey:=2, sName:='enum3'),
		(nKey:=3, sName:='enum4')
	];
END_VAR

fbIngestionConfig(sAssetName := 'Unit-Test-Asset');
Nominal();
EndpointMessageTooBig();
NullArguments();
ConfigParamsExceeded();

METHOD ConfigParamsExceeded : REFERENCE TO FB_Test

VAR
	pFlow1 : POINTER TO ST_FlowConfig;
	pChannel : POINTER TO ST_ChannelConfig;
	sJsonBuffer : STRING(1024);
	stMsg : _ST_SiftMessage;
	stErr : ST_SiftError;
	i,j : UDINT;
END_VAR
// Test creating flows and channels after exceeding the limit.
TEST('CreateIngestionConfig ConfigParamsExceeded');

fbIngestionConfig.ClearIngestionConfig();

pFlow1 := fbIngestionConfig.CreateFlowConfig(sName := 'flow_1');
AssertTrue(pFlow1 <> 0, Message := 'flow_1 was not created successfully');

FOR i := 1 TO SiftClientParameters.MAX_NUM_FLOWS - 1 DO
	AssertTrue(fbIngestionConfig.CreateFlowConfig(sName := 'flow')  <> 0,
			   Message := 'failed to create additional flows');
END_FOR
AssertTrue(fbIngestionConfig.CreateFlowConfig(sName := 'flow') = 0,
		   Message := 'should have exceeded flow capacity');


FOR i := 1 TO SiftClientParameters.MAX_NUM_CHANNELS_PER_FLOW DO
	pChannel := fbIngestionConfig.CreateChannelConfig(pFlowConfig := pFlow1, 
													  sName:='channel',
													  eDataType:=E_ChannelDataType.String_, 
													  sDescription:='A double channel channel', 
													  sUnit:='count');
	AssertTrue(pChannel <> 0, Message := 'channel was not created successfully');	
END_FOR
pChannel := fbIngestionConfig.CreateChannelConfig(pFlowConfig := pFlow1, 
												  sName:='channel',
												  eDataType:=E_ChannelDataType.Double, 
												  sDescription:='A double channel channel', 
												  sUnit:='count');
AssertTrue(pChannel = 0, Message := 'should have exceeded channel capacity');

AssertFalse(fbIngestionConfig.Validate(), 
			Message := 'ingestion config validation should have failed');

TEST_FINISHED();
END_METHOD

METHOD EndpointMessageTooBig : REFERENCE TO FB_Test
VAR_INPUT
END_VAR

VAR
	pFlow1 : POINTER TO ST_FlowConfig;
	pChannel : POINTER TO ST_ChannelConfig;
	sJsonBuffer : STRING(10);
	stMsg : _ST_SiftMessage;
	stErr : ST_SiftError;
	pos : INT;
END_VAR
// Test creating a message that too big to fit in the JsonBuffer.
TEST('CreateIngestionConfig MessageTooBig');

fbIngestionConfig.ClearIngestionConfig();

pFlow1 := fbIngestionConfig.CreateFlowConfig(sName := 'flow_1');
AssertTrue(pFlow1 <> 0, Message := 'flow_1 was not created successfully');

pChannel := fbIngestionConfig.CreateChannelConfig(pFlowConfig := pFlow1, 
									  sName:='longer_than_10_chars',
									  eDataType:=E_ChannelDataType.Double, 
									  sDescription:='A double channel channel', 
									  sUnit:='count');
AssertTrue(pChannel <> 0, Message := 'channel was not created successfully');

stErr := _F_CreateIngestionConfigMessage(stIngestionConfig := fbIngestionConfig.stIngestionConfig, 
							    stMsg := stMsg, 
								pJsonBuffer := ADR(sJsonBuffer), 
								SIZEOF(sJsonBuffer));
								
AssertTrue(stErr.bError, Message := 'CreateIngestionConfigMessage should have returned an error');

pos := FIND(STR1 := stErr.sReason, STR2 := 'JSON msg too large');
AssertTrue(pos <> 0, Message := 'incorrect error string');

TEST_FINISHED();
END_METHOD

METHOD Nominal : REFERENCE TO FB_Test
VAR_INPUT
END_VAR

VAR 
	pFlow1 : POINTER TO ST_FlowConfig;
	pFlow2 : POINTER TO ST_FlowConfig;	
	pChannel : POINTER TO ST_ChannelConfig;
	
	sJsonBuffer : STRING(1500);
	stMsg : _ST_SiftMessage;
	stErr : ST_SiftError;
	
	sExpectedJson : STRING(1500) := '{"endpoint":"create_ingestion_config","data":{"assetName":"Unit-Test-Asset","flows":[{"name":"flow_1","channels":[{"name":"test_channel_1","unit":"count","description":"An enum channel","dataType":"CHANNEL_DATA_TYPE_ENUM","enumTypes":[{"name":"enum1","key":0},{"name":"enum2","key":1},{"name":"enum3","key":2},{"name":"enum4","key":3}]},{"name":"test_channel_2","unit":"a","description":"A bool channel","dataType":"CHANNEL_DATA_TYPE_BOOL","enumTypes":[]},{"name":"test_channel_3","unit":"b","description":"A double channel","dataType":"CHANNEL_DATA_TYPE_DOUBLE","enumTypes":[]},{"name":"test_channel_4","unit":"c","description":"A float channel","dataType":"CHANNEL_DATA_TYPE_FLOAT","enumTypes":[]},{"name":"test_channel_5","unit":"d","description":"A int32 channel","dataType":"CHANNEL_DATA_TYPE_INT_32","enumTypes":[]}]},{"name":"flow_2","channels":[{"name":"test_channel_6","unit":"e","description":"A int64 channel","dataType":"CHANNEL_DATA_TYPE_INT_64","enumTypes":[]},{"name":"test_channel_7","unit":"f","description":"A string channel","dataType":"CHANNEL_DATA_TYPE_STRING","enumTypes":[]},{"name":"test_channel_8","unit":"g","description":"A uint32 channel","dataType":"CHANNEL_DATA_TYPE_UINT_32","enumTypes":[]},{"name":"test_channel_9","unit":"h","description":"A uint64 channel","dataType":"CHANNEL_DATA_TYPE_UINT_64","enumTypes":[]}]}]}}';
END_VAR
// Test creating a nominal ingestion config message.
TEST('CreateIngestionConfig Nominal');

fbIngestionConfig.ClearIngestionConfig();

pFlow1 := fbIngestionConfig.CreateFlowConfig(sName := 'flow_1');
AssertTrue(pFlow1 <> 0, Message := 'flow_1 was not created successfully');

pChannel := fbIngestionConfig.CreateChannelConfig(pFlowConfig := pFlow1, 
													  sName:='test_channel_1', 
													  eDataType:=E_ChannelDataType.Enum, 
													  sDescription:='An enum channel', 
													  sUnit:='count');
AssertTrue(pChannel <> 0, Message := 'enum channel was not created successfully');

AssertTrue(fbIngestionConfig.InitEnumTypes(pChannel, aEnums),
	       Message := 'enum were not initialized correctly');

AssertEquals_UDINT(Expected := aEnums[1].nKey,
				   Actual := pChannel^.aEnumTypes[0].nKey,
				   Message := 'enum 1 key doesnt match');
AssertEquals_UDINT(Expected := aEnums[2].nKey,
				   Actual := pChannel^.aEnumTypes[1].nKey,
				   Message := 'enum 2 key doesnt match');
AssertEquals_UDINT(Expected := aEnums[3].nKey,
				   Actual := pChannel^.aEnumTypes[2].nKey,
				   Message := 'enum 3 key doesnt match');
AssertEquals_UDINT(Expected := aEnums[4].nKey,
				   Actual := pChannel^.aEnumTypes[3].nKey,
				   Message := 'enum 4 key doesnt match');
AssertEquals_STRING(Expected := aEnums[1].sName,
				   Actual := pChannel^.aEnumTypes[0].sName,
				   Message := 'enum 1 name doesnt match');
AssertEquals_STRING(Expected := aEnums[2].sName,
				   Actual := pChannel^.aEnumTypes[1].sName,
				   Message := 'enum 2 name doesnt match');
AssertEquals_STRING(Expected := aEnums[3].sName,
				   Actual := pChannel^.aEnumTypes[2].sName,
				   Message := 'enum 3 name doesnt match');
AssertEquals_STRING(Expected := aEnums[4].sName,
				   Actual := pChannel^.aEnumTypes[3].sName,
				   Message := 'enum 4 name doesnt match');
				   

pChannel := fbIngestionConfig.CreateChannelConfig(pFlowConfig := pFlow1, 
													  sName:='test_channel_2', 
													  eDataType:=E_ChannelDataType.Bool_, 
													  sDescription:='A bool channel', 
													  sUnit:='a');
AssertTrue(pChannel <> 0, Message := 'bool channel was not created successfully');

pChannel := fbIngestionConfig.CreateChannelConfig(pFlowConfig := pFlow1, 
													  sName:='test_channel_3', 
													  eDataType:=E_ChannelDataType.Double, 
													  sDescription:='A double channel', 
													  sUnit:='b');
AssertTrue(pChannel <> 0, Message := 'double channel was not created successfully');

pChannel := fbIngestionConfig.CreateChannelConfig(pFlowConfig := pFlow1, 
													  sName:='test_channel_4', 
													  eDataType:=E_ChannelDataType.Float, 
													  sDescription:='A float channel', 
													  sUnit:='c');
AssertTrue(pChannel <> 0, Message := 'float channel was not created successfully');

pChannel := fbIngestionConfig.CreateChannelConfig(pFlowConfig := pFlow1, 
													  sName:='test_channel_5', 
													  eDataType:=E_ChannelDataType.Int32, 
													  sDescription:='A int32 channel', 
													  sUnit:='d');
AssertTrue(pChannel <> 0, Message := 'int32 channel was not created successfully');

pFlow2 := fbIngestionConfig.CreateFlowConfig(sName := 'flow_2');
AssertTrue(pFlow2 <> 0, Message := 'flow_2 was not created successfully');
pChannel := fbIngestionConfig.CreateChannelConfig(pFlowConfig := pFlow2, 
													  sName:='test_channel_6', 
													  eDataType:=E_ChannelDataType.Int64, 
													  sDescription:='A int64 channel', 
													  sUnit:='e');
AssertTrue(pChannel <> 0, Message := 'int64 channel was not created successfully');

pChannel := fbIngestionConfig.CreateChannelConfig(pFlowConfig := pFlow2, 
													  sName:='test_channel_7', 
													  eDataType:=E_ChannelDataType.String_, 
													  sDescription:='A string channel', 
													  sUnit:='f');
AssertTrue(pChannel <> 0, Message := 'string channel was not created successfully');

pChannel := fbIngestionConfig.CreateChannelConfig(pFlowConfig := pFlow2, 
													  sName:='test_channel_8', 
													  eDataType:=E_ChannelDataType.Uint32, 
													  sDescription:='A uint32 channel', 
													  sUnit:='g');
AssertTrue(pChannel <> 0, Message := 'uint32 channel was not created successfully');

pChannel := fbIngestionConfig.CreateChannelConfig(pFlowConfig := pFlow2, 
													  sName:='test_channel_9', 
													  eDataType:=E_ChannelDataType.Uint64, 
													  sDescription:='A uint64 channel', 
													  sUnit:='h');
AssertTrue(pChannel <> 0, Message := 'uint64 channel was not created successfully');

stErr := _F_CreateIngestionConfigMessage(stIngestionConfig := fbIngestionConfig.stIngestionConfig, 
							    stMsg := stMsg, 
								pJsonBuffer := ADR(sJsonBuffer), 
								SIZEOF(sJsonBuffer));
								
AssertFalse(stErr.bError, Message := 'error creating ingestion config message');
AssertEquals_STRING(Expected := sExpectedJson, 
				    Actual := sJsonBuffer, 
					Message := 'bad ingestion config was created');


TEST_FINISHED();
END_METHOD

METHOD NullArguments : REFERENCE TO FB_Test
VAR
	pFlow1 : POINTER TO ST_FlowConfig;
	pChannel : POINTER TO ST_ChannelConfig;
	stMsg : _ST_SiftMessage;
	stErr : ST_SiftError;
	pos : INT;
END_VAR
// Test creating a message with a null buffer.
TEST('CreateIngestionConfig NullArguments');

fbIngestionConfig.ClearIngestionConfig();

pFlow1 := fbIngestionConfig.CreateFlowConfig(sName := 'flow_1');
AssertTrue(pFlow1 <> 0, Message := 'flow_1 was not created successfully');

pChannel := fbIngestionConfig.CreateChannelConfig(pFlowConfig := pFlow1, 
									  sName:='longer_than_10_chars',
									  eDataType:=E_ChannelDataType.Double, 
									  sDescription:='A double channel channel', 
									  sUnit:='count');
AssertTrue(pChannel <> 0, Message := 'channel was not created successfully');

// Test Null JSON buffer
stErr := _F_CreateIngestionConfigMessage(stIngestionConfig := fbIngestionConfig.stIngestionConfig, 
							    stMsg := stMsg, 
								pJsonBuffer := 0, 
								nLength:= 10);
								
AssertTrue(stErr.bError, Message := 'CreateIngestionConfigMessage did not return an error');

pos := FIND(STR1 := stErr.sReason, STR2 := 'null');
AssertTrue(pos <> 0, Message := 'incorrect error string');

// Test Null flow config
pChannel := fbIngestionConfig.CreateChannelConfig(pFlowConfig := 0, 
												  sName:='channel',
												  eDataType:=E_ChannelDataType.Double, 
												  sDescription:='A double channel channel', 
												  sUnit:='count');
AssertTrue(pChannel = 0, Message := 'channel should have failed');

// Test Null channel
AssertFalse(fbIngestionConfig.InitEnumTypes(pChannelConfig := 0, aEnums),
	       Message := 'enum initialization should have failed');

TEST_FINISHED();
END_METHOD

END_FUNCTION_BLOCK

// ---- Tests/FB_CreatePingMessage_Test.TcPOU
FUNCTION_BLOCK FB_CreatePingMessage_Test EXTENDS TcUnit.FB_TestSuite
VAR_INPUT
END_VAR
VAR_OUTPUT
END_VAR
VAR
END_VAR

Nominal();

METHOD Nominal : REFERENCE TO FB_Test
VAR_INPUT
END_VAR
VAR
	pJsonBuffer : POINTER TO STRING(255);
	stMsg : _ST_SiftMessage;
	stErr : ST_SiftError;
	sExpectedJson : STRING(255) := '{"endpoint":"ping","data":{}}';
END_VAR
// Test creating a nominal ping message.
TEST('CreatePingMessage Nominal');

stErr := _F_CreatePingMessage(stMsg := stMsg);
								
AssertFalse(stErr.bError, Message := 'error creating ping message');

pJsonBuffer := ADR(stMsg.aData);
AssertEquals_STRING(Expected := sExpectedJson, 
				    Actual := pJsonBuffer^, 
				    Message := 'bad ping message was created');

TEST_FINISHED();
END_METHOD

END_FUNCTION_BLOCK

// ---- POUs/Private/_F_CreatePingMessage.TcPOU
// Creates a Sift Proxy Protocol "ping" Endpoint Message.
FUNCTION _F_CreatePingMessage
VAR_INPUT
	stMsg : REFERENCE TO _ST_SiftMessage;
END_VAR

VAR
	sPingRequest : STRING(255) := '{}';
END_VAR

VAR_OUTPUT
	stErr : ST_SiftError;
END_VAR

stErr := _F_CreateEndpointMessage(sEndpoint := 'ping', 
                                  pData := ADR(sPingRequest), 
                                  nLength := INT_TO_UDINT(LEN(sPingRequest)), 
                                  nBufferLength := 255, 
                                  stMsg := stMsg);

END_FUNCTION

// ---- Tests/FB_CreateRunMessage_Test.TcPOU
FUNCTION_BLOCK FB_CreateRunMessage_Test EXTENDS TcUnit.FB_TestSuite
VAR_INPUT
END_VAR
VAR_OUTPUT
END_VAR
VAR
	aTags : ARRAY[1..SiftClientParameters.MAX_NUM_TAGS] OF STRING(255) := [
		'tag1',
		'tag2',
		'another tag'
	];
END_VAR

Nominal();
EndpointMessageTooBig();
NullJsonBuffer();

METHOD EndpointMessageTooBig : REFERENCE TO FB_Test
VAR_INPUT
END_VAR

VAR
	sJsonBuffer : STRING(10);
	stMsg : _ST_SiftMessage;
	stErr : ST_SiftError;
	pos : INT;
END_VAR
// Test creating a message that too big to fit in the JsonBuffer.
TEST('CreateRunMessage MessageTooBig');

stErr := _F_CreateRunMessage(sName := 'Test Run Name',
							 sDescription := 'A description', 
							 aTags := aTags,
							 stMsg := stMsg, 
							 pJsonBuffer := ADR(sJsonBuffer), 
							 nLength:= SIZEOF(sJsonBuffer));
								
AssertTrue(stErr.bError, Message := 'CreateRunMessage did not return an error');

pos := FIND(STR1 := stErr.sReason, STR2 := 'JSON msg too large');
AssertTrue(pos <> 0, Message := 'incorrect error string');

TEST_FINISHED();
END_METHOD

METHOD Nominal : REFERENCE TO FB_Test
VAR_INPUT
END_VAR

VAR
	sJsonBuffer : STRING(255);
	stMsg : _ST_SiftMessage;
	stErr : ST_SiftError;
	sExpectedJson : STRING(255) := '{"endpoint":"create_run","data":{"name":"Test Run Name","description":"A description","tags":["tag1","tag2","another tag"]}}';
END_VAR
// Test creating a nominal ping message.
TEST('CreateRunMessage Nominal');

stErr := _F_CreateRunMessage(sName := 'Test Run Name',
							 sDescription := 'A description', 
							 aTags := aTags,
							 stMsg := stMsg, 
							 pJsonBuffer := ADR(sJsonBuffer), 
							 nLength:= SIZEOF(sJsonBuffer));
								
AssertFalse(stErr.bError, Message := 'error creating run message');
AssertEquals_STRING(Expected := sExpectedJson, 
				    Actual := sJsonBuffer, 
					Message := 'bad ingestion config was created');


TEST_FINISHED();
END_METHOD

METHOD NullJsonBuffer : REFERENCE TO FB_Test
VAR
	stMsg : _ST_SiftMessage;
	stErr : ST_SiftError;
	pos : INT;
END_VAR
// Test creating a message with a null buffer.
TEST('CreateRunMessage NullJsonBuffer');

stErr := _F_CreateRunMessage(sName := 'Test Run Name',
							 sDescription := 'A description', 
							 aTags := aTags,
							 stMsg := stMsg, 
							 pJsonBuffer := 0, 
							 nLength:= 10);
								
AssertTrue(stErr.bError, Message := 'CreateRunMessage did not return an error');

pos := FIND(STR1 := stErr.sReason, STR2 := 'null');
AssertTrue(pos <> 0, Message := 'incorrect error string');

TEST_FINISHED();
END_METHOD

END_FUNCTION_BLOCK

// ---- POUs/Private/_F_CreateRunMessage.TcPOU
// Creates a Sift Proxy Protocol "create_run" Endpoint Message.
FUNCTION _F_CreateRunMessage
VAR_INPUT
	sName : STRING(255);
	sDescription : STRING(255);
	aTags : ARRAY[0..SiftClientParameters.MAX_NUM_TAGS - 1] OF STRING(255);
	stMsg : REFERENCE TO _ST_SiftMessage;
	pJsonBuffer : POINTER TO BYTE;
	nLength : UDINT;
END_VAR

VAR
	fbJson : FB_JsonSaxWriter;
	i : UDINT;
	nBytes : UDINT;
	pJsonString: POINTER TO STRING;
END_VAR

VAR_OUTPUT
	stErr : ST_SiftError;
END_VAR

IF pJsonBuffer = 0 THEN
	stErr.bError := TRUE;
	stErr.nErrId := GVL_SIFT.NULL_JSON_POINTER;
	stErr.sReason := 'The JSON buffer is null';
	RETURN;
END_IF

fbJson.StartObject();

fbJson.AddKey('name');
fbJson.AddString(sName);

fbJson.AddKey('description');
fbJson.AddString(sDescription);

fbJson.AddKey('tags');
fbJson.StartArray();
FOR i := 1 TO SiftClientParameters.MAX_NUM_TAGS DO
	IF LEN(aTags[i-1]) > 0 THEN
		 fbJson.AddString(aTags[i-1]);
	END_IF
END_FOR
fbJson.EndArray();

fbJson.EndObject();

pJsonString := pJsonBuffer;
nBytes := fbJson.CopyDocument(pJsonString^, nLength);
IF nBytes = 0 THEN
	stErr.nErrId := GVL_SIFT.JSON_CAPACITY_REACHED;
	stErr.bError := TRUE;
	stErr.sReason := CONCAT(
		CONCAT('JSON msg too large: ', UDINT_TO_STRING(fbJson.GetDocumentLength())),
		' endpoint=create_run',
	);
	RETURN;
END_IF

stErr := _F_CreateEndpointMessage(sEndpoint:='create_run', 
								  pData:=pJsonString, 
								  nLength:=nBytes-1, 
                                  nBufferLength := nLength, 
                                  stMsg:=stMsg);

END_FUNCTION

// ---- Tests/FB_SiftError_Test.TcPOU
FUNCTION_BLOCK FB_SiftError_Test EXTENDS TcUnit.FB_TestSuite
VAR_INPUT
END_VAR
VAR_OUTPUT
END_VAR
VAR
END_VAR

Responses();

METHOD Responses : REFERENCE TO FB_Test
VAR
	fbJson : FB_JsonDomParser;
	sResponse : STRING(GVL_SIFT.MAX_JSON_RESPONSE_SIZE);
	jsonDoc : SJsonValue;
	stErr : ST_SiftError;
END_VAR
TEST('SiftError Responses');

// Test 1: Nominal response
sResponse := '{
	"status": true,
	"data": {}
}';
jsonDoc := fbJson.ParseDocument(sResponse);
AssertTrue(_F_IsSuccessfulResponse(jsonDoc), Message := 'failed to parse successful response');

// Test 2: Failure response
sResponse := '{
	"status": false,
	"data": {}
}';
jsonDoc := fbJson.ParseDocument(sResponse);
AssertFalse(_F_IsSuccessfulResponse(jsonDoc), Message := 'failed to parse failure response');

// Test 3: Failure response with reason
sResponse := '{
	"status": false,
	"data": {
		"reason": "this is the reason for the error"
	}
}';
jsonDoc := fbJson.ParseDocument(sResponse);
AssertTrue(_F_SetSiftError(jsonDoc, stErr), Message := 'failed to parse error');
AssertTrue(stErr.bError, Message := 'error flag not set');
AssertEquals_STRING(Expected := 'this is the reason for the error',
					Actual := stErr.sReason,
					Message := 'reason does not match');
					
// Test 4: 'status' spelled wrong
sResponse := '{
	"status_": false,
	"data": {}
}';
jsonDoc := fbJson.ParseDocument(sResponse);
AssertFalse(_F_SetSiftError(jsonDoc, stErr), Message := 'failed to handle status typo');

// Test 5: 'response' spelled wrong
sResponse := '{
	"status": false,
	"response_": {}
}';
jsonDoc := fbJson.ParseDocument(sResponse);
AssertFalse(_F_SetSiftError(jsonDoc, stErr), Message := 'failed to handle response typo');

// Test 6: 'reason' spelled wrong
sResponse := '{
	"status": false,
	"data": {
		"reason_": "this is the reason for the error"
	}
}';
jsonDoc := fbJson.ParseDocument(sResponse);
AssertFalse(_F_SetSiftError(jsonDoc, stErr), Message := 'failed to handle reason typo');

TEST_FINISHED();
END_METHOD

END_FUNCTION_BLOCK

// ---- Tests/FB_CreateDataMessage_Test.TcPOU
FUNCTION_BLOCK FB_CreateDataMessage_Test EXTENDS TcUnit.FB_TestSuite
VAR_INPUT
END_VAR
VAR_OUTPUT
END_VAR
VAR
	pFlow1 : POINTER TO ST_FlowConfig;
	pFlow2 : POINTER TO ST_FlowConfig;	
	pEmptyFlow : POINTER TO ST_FlowConfig;	
	pEnumChannel : POINTER TO ST_ChannelConfig;
	pBoolChannel : POINTER TO ST_ChannelConfig;
	pDoubleChannel : POINTER TO ST_ChannelConfig;
	pFloatChannel : POINTER TO ST_ChannelConfig;
	pInt32Channel : POINTER TO ST_ChannelConfig;
	pInt64Channel : POINTER TO ST_ChannelConfig;
	pStringChannel : POINTER TO ST_ChannelConfig;
	pUint32Channel : POINTER TO ST_ChannelConfig;
	pUint64Channel : POINTER TO ST_ChannelConfig;
	aEnums : ARRAY[1..SiftClientParameters.MAX_NUM_ENUMS_PER_CHANNEL] OF ST_EnumType := [
		(nKey:=0, sName:='enum1'),
		(nKey:=1, sName:='enum2'),
		(nKey:=2, sName:='enum3'),
		(nKey:=3, sName:='enum4')
	];

	aRawBuf : ARRAY[0..SiftClientParameters.MAX_PACKET_SIZE - 1] OF BYTE;
	fbWriter : _FB_BufferWriter := (pRawBuf := ADR(aRawBuf), nSize := SIZEOF(aRawBuf));

	fbIngest : FB_IngestService;	
	fbIngestionConfig : FB_IngestionConfigService;
END_VAR

fbIngestionConfig.ClearIngestionConfig();

pFlow1 := fbIngestionConfig.CreateFlowConfig(sName := 'flow_1');
AssertTrue(pFlow1 <> 0, Message := 'flow_1 was not created successfully');

pEnumChannel := fbIngestionConfig.CreateChannelConfig(pFlowConfig := pFlow1, 
													  sName:='test_channel_1', 
													  eDataType:=E_ChannelDataType.Enum, 
													  sDescription:='An enum channel', 
													  sUnit:='count');
AssertTrue(pEnumChannel <> 0, Message := 'enum channel was not created successfully');

AssertTrue(fbIngestionConfig.InitEnumTypes(pEnumChannel, aEnums),
	       Message := 'enum were not initialized correctly');

pBoolChannel := fbIngestionConfig.CreateChannelConfig(pFlowConfig := pFlow1, 
													  sName:='test_channel_2', 
													  eDataType:=E_ChannelDataType.Bool_, 
													  sDescription:='A bool channel', 
													  sUnit:='a');
AssertTrue(pBoolChannel <> 0, Message := 'bool channel was not created successfully');

pDoubleChannel := fbIngestionConfig.CreateChannelConfig(pFlowConfig := pFlow1, 
													  sName:='test_channel_3', 
													  eDataType:=E_ChannelDataType.Double, 
													  sDescription:='A double channel', 
													  sUnit:='b');
AssertTrue(pDoubleChannel <> 0, Message := 'double channel was not created successfully');

pFloatChannel := fbIngestionConfig.CreateChannelConfig(pFlowConfig := pFlow1, 
													  sName:='test_channel_4', 
													  eDataType:=E_ChannelDataType.Float, 
													  sDescription:='A float channel', 
													  sUnit:='c');
AssertTrue(pFloatChannel <> 0, Message := 'float channel was not created successfully');

pInt32Channel := fbIngestionConfig.CreateChannelConfig(pFlowConfig := pFlow1, 
													  sName:='test_channel_5', 
													  eDataType:=E_ChannelDataType.Int32, 
													  sDescription:='A int32 channel', 
													  sUnit:='d');
AssertTrue(pInt32Channel <> 0, Message := 'int32 channel was not created successfully');

pFlow2 := fbIngestionConfig.CreateFlowConfig(sName := 'flow_2');
AssertTrue(pFlow2 <> 0, Message := 'flow_2 was not created successfully');
pInt64Channel := fbIngestionConfig.CreateChannelConfig(pFlowConfig := pFlow2, 
													  sName:='test_channel_6', 
													  eDataType:=E_ChannelDataType.Int64, 
													  sDescription:='A int64 channel', 
													  sUnit:='e');
AssertTrue(pInt64Channel <> 0, Message := 'int64 channel was not created successfully');

pStringChannel := fbIngestionConfig.CreateChannelConfig(pFlowConfig := pFlow2, 
													  sName:='test_channel_7', 
													  eDataType:=E_ChannelDataType.String_, 
													  sDescription:='A string channel', 
													  sUnit:='f');
AssertTrue(pStringChannel <> 0, Message := 'string channel was not created successfully');

pUint32Channel := fbIngestionConfig.CreateChannelConfig(pFlowConfig := pFlow2, 
													  sName:='test_channel_8', 
													  eDataType:=E_ChannelDataType.Uint32, 
													  sDescription:='A uint32 channel', 
													  sUnit:='g');
AssertTrue(pUint32Channel <> 0, Message := 'uint32 channel was not created successfully');

pUint64Channel := fbIngestionConfig.CreateChannelConfig(pFlowConfig := pFlow2, 
													  sName:='test_channel_9', 
													  eDataType:=E_ChannelDataType.Uint64, 
													  sDescription:='A uint64 channel', 
													  sUnit:='h');
AssertTrue(pUint64Channel <> 0, Message := 'uint64 channel was not created successfully');

pEmptyFlow := fbIngestionConfig.CreateFlowConfig(sName := 'flow_3_empty');
AssertTrue(pEmptyFlow <> 0, Message := 'flow_3_empty was not created successfully');

Nominal();
InvalidWrites();

METHOD InvalidWrites : REFERENCE TO FB_Test
VAR
	aRawBufSmall : ARRAY[0..10] OF BYTE;
	fbWriterSmall : _FB_BufferWriter := (pRawBuf := ADR(aRawBufSmall), nSize := SIZEOF(aRawBufSmall));
	stTimestamp : _ST_Timestamp;
	nBytes: UDINT;
END_VAR
TEST('CreateDataMessage InvalidWrites');  

// Null Flow
AssertTrue(_F_CreateDataMessage(fbWriter := fbWriterSmall, 
			    			   pFlowConfig := 0, 
							   sRunId := 'test-run-id',
							   stTimestamp := stTimestamp) = 0,
			Message := 'should error on null flow');

// Small buffer
AssertTrue(_F_CreateDataMessage(fbWriter := fbWriterSmall, 
			    			   pFlowConfig := pFlow1, 
							   sRunId := 'test-run-id',
							   stTimestamp := stTimestamp) = 0,
			Message := 'should error on small flow');
							   
TEST_FINISHED();
END_METHOD

METHOD Nominal : REFERENCE TO FB_Test
VAR_INPUT
END_VAR

VAR 
	nEnumTestValue : UDINT := 10;
	bBoolTestValue : BOOL := TRUE;
	fDoubleTestValue : LREAL := 1.2345;
	fFloatTestValue : REAL := 9.8765;
	nInt32TestValue : DINT := 12345;
	nInt64TestValue : LINT := -12232423;
	sStringTestValue : STRING(255) := 'Test string value';
	nUInt32TestValue : UDINT := 4893573;
	nUInt64TestValue : ULINT := 1249864785;
	sRunId : STRING := 'test-run-id';
	
	stMsg : _ST_SiftMessage;
	stErr : ST_SiftError;
	stTimestamp : _ST_Timestamp;
	nBytes : UDINT;
	nValuesOffset : UDINT;
	
	bTmpBool : BOOL;
	fTmpDouble : LREAL;
	fTmpFloat : REAL;
	nTmpUdint : UDINT;
	nTmpUlint : ULINT;
	nTmpLint : LINT;
	nTmpDint : DINT;
	pTmpString : POINTER TO STRING;
END_VAR
// Test creating a nominal data message
TEST('CreateDataMessage Nominal');

AssertTrue(SetChannelValue(pChannel := pEnumChannel, nEnumTestValue),
           Message := 'the enum value was not set correctly');
AssertTrue(SetChannelValue(pChannel := pBoolChannel, bBoolTestValue),
           Message := 'the bool value was not set correctly');
AssertTrue(SetChannelValue(pChannel := pDoubleChannel, fDoubleTestValue),
           Message := 'the double value was not set correctly');
AssertTrue(SetChannelValue(pChannel := pFloatChannel, fFloatTestValue),
           Message := 'the float value was not set correctly');
AssertTrue(SetChannelValue(pChannel := pInt32Channel, nInt32TestValue),
           Message := 'the int32 value was not set correctly');
AssertTrue(SetChannelValue(pChannel := pInt64Channel, nInt64TestValue),
           Message := 'the int64 value was not set correctly');
AssertTrue(SetChannelValue(pChannel := pStringChannel, sStringTestValue),
           Message := 'the string value was not set correctly');
AssertTrue(SetChannelValue(pChannel := pUint32Channel, nUInt32TestValue),
           Message := 'the uint32 value was not set correctly');
AssertTrue(SetChannelValue(pChannel := pUint64Channel, nUInt64TestValue),
           Message := 'the uint64 value was not set correctly');
		   
stTimestamp.nSeconds := 1234567;		   
stTimestamp.nNanoseconds := 65432;		   

// Flow 1	  
nBytes := _F_CreateDataMessage(fbWriter := fbWriter, 
			    			   pFlowConfig := pFlow1, 
							   sRunId := sRunId,
							   stTimestamp := stTimestamp);
 
MEMCPY(ADR(nTmpUdint), ADR(aRawBuf[0]), 4);
AssertEquals_UDINT(Expected := GVL_SIFT.SYNC_WORD,
				   Actual := nTmpUdint,
				   Message := 'sync word did not match');
				   
AssertEquals_BYTE(Expected := GVL_SIFT.DATA_MESSAGE_TYPE,
				  Actual := aRawBuf[GVL_SIFT.MESSAGE_TYPE_INDEX],
				  Message := 'incorrect message type');
				  
MEMCPY(ADR(nTmpUdint), ADR(aRawBuf[GVL_SIFT.MESSGE_LENGTH_INDEX]), 4);
AssertEquals_UDINT(Expected := nBytes,
				   Actual := nTmpUdint,
				   Message := 'incorrect message length');
				   
MEMCPY(ADR(nTmpLint), ADR(aRawBuf[GVL_SIFT.HEADER_LENGTH]), 8);
AssertEquals_LINT(Expected := stTimestamp.nSeconds,
				   Actual := nTmpLint,
				   Message := 'incorrect timestamp (seconds)');
				   
MEMCPY(ADR(nTmpDint), ADR(aRawBuf[GVL_SIFT.HEADER_LENGTH+8]), 4);
AssertEquals_LINT(Expected := stTimestamp.nNanoseconds,
				   Actual := nTmpDint,
				   Message := 'incorrect timestamp (nanoseconds)');

pTmpString := ADR(aRawBuf[GVL_SIFT.HEADER_LENGTH+12]);
AssertEquals_STRING(Expected := pFlow1^.sName,
				    Actual := pTmpString^,
				    Message := 'incorrect flow');
					
pTmpString := ADR(aRawBuf[GVL_SIFT.HEADER_LENGTH+12 + DINT_TO_UDINT(LEN(pFlow1^.sName)) + 1]);
AssertEquals_STRING(Expected := sRunId,
				    Actual := pTmpString^,
				    Message := 'incorrect run id');
					
nValuesOffset := GVL_SIFT.HEADER_LENGTH+12 + DINT_TO_UDINT(LEN(pFlow1^.sName)) + 1 + DINT_TO_UDINT(LEN(sRunId)) + 1;
		   
MEMCPY(ADR(nTmpUdint), ADR(aRawBuf[nValuesOffset]), SIZEOF(nEnumTestValue));
AssertEquals_UDINT(Expected := nEnumTestValue,
				   Actual := nTmpUdint,
				   Message := 'incorrect enum value in message');
nValuesOffset := nValuesOffset + SIZEOF(nEnumTestValue);

MEMCPY(ADR(bTmpBool), ADR(aRawBuf[nValuesOffset]), SIZEOF(bBoolTestValue));
AssertEquals_BOOL(Expected := bBoolTestValue,
				   Actual := bTmpBool,
				   Message := 'incorrect bool value in message');
nValuesOffset := nValuesOffset + SIZEOF(bBoolTestValue);

MEMCPY(ADR(fTmpDouble), ADR(aRawBuf[nValuesOffset]), SIZEOF(fDoubleTestValue));
AssertEquals_LREAL(Expected := fDoubleTestValue,
				   Actual := fTmpDouble,
				   Delta := 0,
				   Message := 'incorrect double value in message');
nValuesOffset := nValuesOffset + SIZEOF(fDoubleTestValue);
				   
MEMCPY(ADR(fTmpFloat), ADR(aRawBuf[nValuesOffset]), SIZEOF(fFloatTestValue));
AssertEquals_LREAL(Expected := fFloatTestValue,
				   Actual := fTmpFloat,
				   Delta := 0,
				   Message := 'incorrect float value in message');
nValuesOffset := nValuesOffset + SIZEOF(fFloatTestValue);

MEMCPY(ADR(nTmpDint), ADR(aRawBuf[nValuesOffset]), SIZEOF(nInt32TestValue));
AssertEquals_DINT(Expected := nInt32TestValue,
				   Actual := nTmpDint,
				   Message := 'incorrect int32 value in message');
nValuesOffset := nValuesOffset + SIZEOF(nInt32TestValue);

// Flow 2
fbWriter.SetOffset(0);

// Test empty run
sRunId := '';

nBytes := _F_CreateDataMessage(fbWriter := fbWriter, 
			    			   pFlowConfig := pFlow2, 
							   sRunId := sRunId,
							   stTimestamp := stTimestamp);
 
MEMCPY(ADR(nTmpUdint), ADR(aRawBuf[0]), 4);
AssertEquals_UDINT(Expected := GVL_SIFT.SYNC_WORD,
				   Actual := nTmpUdint,
				   Message := 'sync word did not match');
				   
AssertEquals_BYTE(Expected := GVL_SIFT.DATA_MESSAGE_TYPE,
				  Actual := aRawBuf[GVL_SIFT.MESSAGE_TYPE_INDEX],
				  Message := 'incorrect message type');
				  
MEMCPY(ADR(nTmpUdint), ADR(aRawBuf[GVL_SIFT.MESSGE_LENGTH_INDEX]), 4);
AssertEquals_UDINT(Expected := nBytes,
				   Actual := nTmpUdint,
				   Message := 'incorrect message length');
				   
MEMCPY(ADR(nTmpLint), ADR(aRawBuf[GVL_SIFT.HEADER_LENGTH]), 8);
AssertEquals_LINT(Expected := stTimestamp.nSeconds,
				   Actual := nTmpLint,
				   Message := 'incorrect timestamp (seconds)');
				   
MEMCPY(ADR(nTmpDint), ADR(aRawBuf[GVL_SIFT.HEADER_LENGTH+8]), 4);
AssertEquals_LINT(Expected := stTimestamp.nNanoseconds,
				   Actual := nTmpDint,
				   Message := 'incorrect timestamp (nanoseconds)');

pTmpString := ADR(aRawBuf[GVL_SIFT.HEADER_LENGTH+12]);
AssertEquals_STRING(Expected := pFlow2^.sName,
				    Actual := pTmpString^,
				    Message := 'incorrect flow');
					
pTmpString := ADR(aRawBuf[GVL_SIFT.HEADER_LENGTH+12 + DINT_TO_UDINT(LEN(pFlow2^.sName)) + 1]);
AssertEquals_STRING(Expected := sRunId,
				    Actual := pTmpString^,
				    Message := 'incorrect run id');
					
nValuesOffset := GVL_SIFT.HEADER_LENGTH+12 + DINT_TO_UDINT(LEN(pFlow2^.sName)) + 1 + DINT_TO_UDINT(LEN(sRunId)) + 1;
		   
MEMCPY(ADR(nTmpLint), ADR(aRawBuf[nValuesOffset]), SIZEOF(nInt64TestValue));
AssertEquals_LINT(Expected := nInt64TestValue,
				   Actual := nTmpLint,
				   Message := 'incorrect int64 value in message');
nValuesOffset := nValuesOffset + SIZEOF(nInt64TestValue);

pTmpString := ADR(aRawBuf[nValuesOffset]);
AssertEquals_STRING(Expected := sStringTestValue,
				    Actual := pTmpString^,
				    Message := 'incorrect string value in message');
nValuesOffset := nValuesOffset + DINT_TO_UDINT(LEN(sStringTestValue)) + 1;

MEMCPY(ADR(nTmpUdint), ADR(aRawBuf[nValuesOffset]), SIZEOF(nUInt32TestValue));
AssertEquals_UDINT(Expected := nUInt32TestValue,
				   Actual := nTmpUdint,
				   Message := 'incorrect uint32 value in message');
nValuesOffset := nValuesOffset + SIZEOF(nUInt32TestValue);

MEMCPY(ADR(nTmpUlint), ADR(aRawBuf[nValuesOffset]), SIZEOF(nUInt64TestValue));
AssertEquals_ULINT(Expected := nUInt64TestValue,
				   Actual := nTmpUlint,
				   Message := 'incorrect uint64 value in message');
nValuesOffset := nValuesOffset + SIZEOF(nUInt64TestValue);

// Empty Flow
fbWriter.SetOffset(0);
nBytes := _F_CreateDataMessage(fbWriter := fbWriter, 
			    			   pFlowConfig := pEmptyFlow, 
							   sRunId := sRunId,
							   stTimestamp := stTimestamp);
							   
MEMCPY(ADR(nTmpUdint), ADR(aRawBuf[0]), 4);
AssertEquals_UDINT(Expected := GVL_SIFT.SYNC_WORD,
				   Actual := nTmpUdint,
				   Message := 'sync word did not match');
				   
AssertEquals_BYTE(Expected := GVL_SIFT.DATA_MESSAGE_TYPE,
				  Actual := aRawBuf[GVL_SIFT.MESSAGE_TYPE_INDEX],
				  Message := 'incorrect message type');
				  
MEMCPY(ADR(nTmpUdint), ADR(aRawBuf[GVL_SIFT.MESSGE_LENGTH_INDEX]), 4);
AssertEquals_UDINT(Expected := nBytes,
				   Actual := nTmpUdint,
				   Message := 'incorrect message length');
				   
MEMCPY(ADR(nTmpLint), ADR(aRawBuf[GVL_SIFT.HEADER_LENGTH]), 8);
AssertEquals_LINT(Expected := stTimestamp.nSeconds,
				   Actual := nTmpLint,
				   Message := 'incorrect timestamp (seconds)');
				   
MEMCPY(ADR(nTmpDint), ADR(aRawBuf[GVL_SIFT.HEADER_LENGTH+8]), 4);
AssertEquals_LINT(Expected := stTimestamp.nNanoseconds,
				   Actual := nTmpDint,
				   Message := 'incorrect timestamp (nanoseconds)');

pTmpString := ADR(aRawBuf[GVL_SIFT.HEADER_LENGTH+12]);
AssertEquals_STRING(Expected := pEmptyFlow^.sName,
				    Actual := pTmpString^,
				    Message := 'incorrect flow');
					
pTmpString := ADR(aRawBuf[GVL_SIFT.HEADER_LENGTH+12 + DINT_TO_UDINT(LEN(pEmptyFlow^.sName)) + 1]);
AssertEquals_STRING(Expected := sRunId,
				    Actual := pTmpString^,
				    Message := 'incorrect run id');

TEST_FINISHED();
END_METHOD

END_FUNCTION_BLOCK

// ---- POUs/Services/FB_IngestService.TcPOU
// Service for ingesting data. This function block should be called on 
// every cycle to continually stream any data stored in the internal buffer.
FUNCTION_BLOCK FB_IngestService
VAR_INPUT
	hSiftClient : REFERENCE TO T_SiftClient;
	sRunId : STRING(255);
	aFlowConfigs : POINTER TO ST_FlowConfig;
END_VAR

VAR_OUTPUT
	bBusy : BOOL; // Set to high while data is being transferred.
	bError : BOOL;
	nErrId : UDINT;
	nMsgsSent : UDINT; // Number of total messages sent to sift_proxy.
	nBufSize : UDINT; // The number of messages in the buffer.
	fBufferUtilization : LREAL; // The percent utilization of the internal buffer.
END_VAR

VAR
	eState : (IDLE, SEND_MESSAGE, SEND_MESSAGE_WAIT, SUCCESS, FAILURE):= IDLE;
	fbSendRingBuffer : FB_MemRingBuffer;
	aSendRingBuffer : ARRAY[0..SiftClientParameters.MAX_PACKET_SIZE - 1] OF BYTE;
	aTmpBuffer : ARRAY[0..SiftClientParameters.MAX_PACKET_SIZE - 1] OF BYTE;
	curOffset : UDINT;
	i : UDINT;
	nCount : UDINT;
END_VAR

nBufSize := fbSendRingBuffer.nCount;
fBufferUtilization := UDINT_TO_LREAL(fbSendRingBuffer.cbSize) / UDINT_TO_LREAL(SiftClientParameters.MAX_PACKET_SIZE);

CASE eState OF
	IDLE:
    	bBusy := FALSE;
		bError := FALSE;
		IF nBufSize > 0 THEN
			nCount := nBufSize;
			eState := SEND_MESSAGE;
			
		END_IF
			
	SEND_MESSAGE:
		bBusy := TRUE;
		bError := FALSE;
		curOffset := 0;
		FOR i := 1 TO nCount DO
			fbSendRingBuffer.A_RemoveHead(pRead := ADR(aTmpBuffer[curOffset]),
										  cbRead := SiftClientParameters.MAX_PACKET_SIZE - curOffset,
										  pBuffer := ADR(aSendRingBuffer),
										  cbBuffer := SiftClientParameters.MAX_PACKET_SIZE);
			IF NOT fbSendRingBuffer.bOk THEN
				eState := FAILURE;
				nErrId := GVL_SIFT.INGEST_RING_BUFFER_REMOVE_ERROR;
				RETURN;
			END_IF
			curOffset := curOffset + fbSendRingBuffer.cbReturn;
		END_FOR
		nCount := 0;
		
		hSiftClient.fbSend(
			hSocket := hSiftClient.fbConnect.hSocket, 
			pSrc := ADR(aTmpBuffer),
			cbLen := curOffset,
			bExecute := TRUE,
		);
		
		eState := SEND_MESSAGE_WAIT;

	SEND_MESSAGE_WAIT:
	    bBusy := TRUE;
		bError := FALSE;
		hSiftClient.fbSend(bExecute := FALSE);
		
		IF hSiftClient.fbSend.bBusy THEN
			RETURN;
		ELSIF hSiftClient.fbSend.bError THEN
			nErrId := hSiftClient.fbSend.nErrId;
			eState := FAILURE;
			RETURN;
		END_IF	
		
		nMsgsSent := nMsgsSent + 1;
		eState := IDLE;
		
	FAILURE:
	    bBusy := FALSE;
		bError := TRUE;
END_CASE

// Writes data from a Flow to the buffer to be sent to Sift.
// This should be called for each time you want to record data
// for a given flow.
METHOD PUBLIC WriteData : BOOL
VAR_INPUT
	pFlowConfig : POINTER TO ST_FlowConfig;
	stTimestamp : _ST_Timestamp;
END_VAR

VAR_OUTPUT
	bError : BOOL;
END_VAR

VAR
	// TODO: This should be allocated on the heap (FB local var);
	aRawBuf : ARRAY[1..SiftClientParameters.MAX_PACKET_SIZE] OF BYTE;
	fbWriter : _FB_BufferWriter := (pRawBuf := ADR(aRawBuf), nSize := SIZEOF(aRawBuf));
	nMsgSize : UDINT;
END_VAR
IF pFlowConfig = 0 THEN
	WriteData := FALSE;
	RETURN;
END_IF

nMsgSize := _F_CreateDataMessage(fbWriter := fbWriter, 
							     pFlowConfig := pFlowConfig, 
								 sRunId := sRunId,
							     stTimestamp := stTimestamp);
IF nMsgSize = 0 THEN
	WriteData := FALSE;
	RETURN;
END_IF

fbSendRingBuffer.A_AddTail(pWrite := ADR(aRawBuf), 
						   cbWrite := nMsgSize + GVL_SIFT.HEADER_LENGTH, 
						   pBuffer := ADR(aSendRingBuffer), 
						   cbBuffer := SiftClientParameters.MAX_PACKET_SIZE);
						   
WriteData := fbSendRingBuffer.bOk;
END_METHOD

END_FUNCTION_BLOCK

// ---- POUs/Private/_F_CreateDataMessage.TcPOU
// Creates a Sift Proxy Protocol Data Message.
FUNCTION _F_CreateDataMessage : UDINT;

VAR_INPUT
	fbWriter : REFERENCE TO _FB_BufferWriter;
	pFlowConfig : POINTER TO ST_FlowConfig;
	sRunId : STRING(255);
	stTimestamp : _ST_Timestamp;
END_VAR

VAR
	stFlowConfig : REFERENCE TO ST_FlowConfig;
	tmpCC : REFERENCE TO ST_ChannelConfig;
	nStrLen : UINT;
	nMsgSize : UDINT;
	i : UDINT;
END_VAR

IF pFlowConfig = 0 THEN
	_F_CreateDataMessage := 0;
	RETURN;
END_IF

stFlowConfig REF= pFlowConfig^;

IF NOT fbWriter.SetOffset(GVL_SIFT.HEADER_LENGTH) THEN
	_F_CreateDataMessage := 0;
	RETURN;
END_IF

(* Timestamp *);
IF NOT fbWriter.Write(ADR(stTimestamp.nSeconds), 8) THEN
		_F_CreateDataMessage := 0;
	RETURN;
END_IF

IF NOT fbWriter.Write(ADR(stTimestamp.nNanoseconds), 4) THEN
		_F_CreateDataMessage := 0;
	RETURN;
END_IF

(* Flow Name *)
nStrLen := INT_TO_UINT(LEN(stFlowConfig.sName));
IF NOT fbWriter.Write(ADR(stFlowConfig.sName), nStrLen) THEN
		_F_CreateDataMessage := 0;
	RETURN;
END_IF
IF NOT fbWriter.WriteByte(0) THEN
		_F_CreateDataMessage := 0;
	RETURN;
END_IF

(* Run ID *)
nStrLen := INT_TO_UINT(LEN(sRunId));
IF NOT fbWriter.Write(ADR(sRunId), nStrLen) THEN
		_F_CreateDataMessage := 0;
	RETURN;
END_IF
IF NOT fbWriter.WriteByte(0) THEN
		_F_CreateDataMessage := 0;
	RETURN;
END_IF

FOR i := 1 TO stFlowConfig.nNumChannelConfigs  BY 1 DO
	tmpCC REF= stFlowConfig.aChannelConfigs[i-1];
	
	CASE tmpCC.eDataType OF
		E_ChannelDataType.Bool_:
			IF NOT fbWriter.Write(ADR(tmpCC.Value.bBool), 1) THEN
				_F_CreateDataMessage := 0;
				RETURN;
			END_IF
	
		E_ChannelDataType.Double:
			IF NOT fbWriter.Write(ADR(tmpCC.Value.fDouble), 8) THEN
				_F_CreateDataMessage := 0;
				RETURN;
			END_IF
			
		E_ChannelDataType.Enum:
			IF NOT fbWriter.Write(ADR(tmpCC.Value.nEnum), 4) THEN
				_F_CreateDataMessage := 0;
				RETURN;
			END_IF
			
		E_ChannelDataType.Float:
			IF NOT fbWriter.Write(ADR(tmpCC.Value.fFloat), 4) THEN
				_F_CreateDataMessage := 0;
				RETURN;
			END_IF
			
		E_ChannelDataType.Int32:
			IF NOT fbWriter.Write(ADR(tmpCC.Value.nInt32), 4) THEN
				_F_CreateDataMessage := 0;
				RETURN;
			END_IF
			
		E_ChannelDataType.Int64:
			IF NOT fbWriter.Write(ADR(tmpCC.Value.nInt64), 8) THEN
				_F_CreateDataMessage := 0;
				RETURN;
			END_IF
			
		E_ChannelDataType.UInt32:
			IF NOT fbWriter.Write(ADR(tmpCC.Value.nInt32), 4) THEN
				_F_CreateDataMessage := 0;
				RETURN;
			END_IF
			
		E_ChannelDataType.UInt64:
			IF NOT fbWriter.Write(ADR(tmpCC.Value.nInt64), 8) THEN
				_F_CreateDataMessage := 0;
				RETURN;
			END_IF
			
		E_ChannelDataType.String_:
			nStrLen := INT_TO_UINT(LEN(tmpCC.Value.sString));
			IF NOT fbWriter.Write(ADR(tmpCC.Value.sString), nStrLen) THEN
				_F_CreateDataMessage := 0;
					RETURN;
			END_IF
			IF NOT fbWriter.WriteByte(0) THEN
				_F_CreateDataMessage := 0;
				RETURN;
			END_IF
	END_CASE

END_FOR

IF NOT fbWriter.WriteAt(0, ADR(GVL_SIFT.SYNC_WORD), 4) THEN
	_F_CreateDataMessage := 0;
	RETURN;
END_IF

IF NOT fbWriter.WriteAt(GVL_SIFT.MESSAGE_TYPE_INDEX, ADR(GVL_SIFT.DATA_MESSAGE_TYPE), 1) THEN
	_F_CreateDataMessage := 0;
	RETURN;
END_IF

nMsgSize := fbWriter.nCurOffset - GVL_SIFT.HEADER_LENGTH;
IF NOT fbWriter.WriteAt(GVL_SIFT.MESSGE_LENGTH_INDEX, ADR(nMsgSize), 4) THEN
	_F_CreateDataMessage := 0;
	RETURN;
END_IF

						   
_F_CreateDataMessage := nMsgSize;

END_FUNCTION

// ---- POUs/FB_SiftClient.TcPOU
// Entry point for the Sift Client. This function block must be initialized successfully
// first before using any of the other services. The function block begins initialization
// on the rising edge of bExecute and completes initialization when bBusy goes low.
FUNCTION_BLOCK FB_SiftClient
VAR_INPUT
	sSiftProxyHost : T_IPv4Addr := GVL_SIFT.SIFT_PROXY_DEFAULT_HOST;
	nSiftProxyPort : UINT       := GVL_SIFT.SIFT_PROXY_DEFAULT_LISTEN_PORT;
	sLogDir : STRING(255);
	
	sGrpcUri : STRING(255);
	sApiKey : STRING(255);
	
	pJsonBuffer : POINTER TO BYTE;
	pJbLength : UDINT;
	
	bExecute : BOOL;
	bStop : BOOL;
END_VAR

VAR_OUTPUT
	hSiftClient : T_SiftClient;
	bBusy : BOOL;
	bError : BOOL;
	nErrId : UDINT;
	nErrMsg : STRING(255);
END_VAR

VAR
    fbAuth : FB_AuthenticateService;	
	fbStartSiftProxy : NT_StartProcess;
	fbGetLocalAmsNetID : FB_GetLocalAmsNetId;
	fbFormat : FB_FormatString;
	nAttempts : UINT;
	startDelay : TON;
	
	eState : (
		IDLE, 
		CLOSE_ALL, 
		CLOSE_ALL_WAIT, 
		CONNECT, 
		CONNECT_WAIT, 
		GET_LOCAL_AMD_NET_ID,
		GET_LOCAL_AMD_NET_ID_WAIT,
		START_SIFT_PROXY, 
		START_SIFT_PROXY_DELAY,
		START_SIFT_PROXY_WAIT,
		AUTHENTICATE,
		AUTHENTICATE_WAIT,
		SUCCESS, 
		FAILURE,
		STOP,
		STOP_WAIT,
	) := IDLE;
END_VAR

CASE eState OF
	IDLE:
	    bBusy := FALSE;
		IF bExecute THEN
			eState := CLOSE_ALL;
		ELSIF bStop THEN
			eState := STOP;
		END_IF

	CLOSE_ALL:
		bBusy := TRUE;
		bError := FALSE;
		hSiftClient.fbCloseAll(bExecute := TRUE);
		nAttempts := 0;
		eState := CLOSE_ALL_WAIT;
		
	CLOSE_ALL_WAIT:
		bBusy := TRUE;
		bError := FALSE;
		hSiftClient.fbCloseAll(bExecute := FALSE);
		
		IF hSiftClient.fbCloseAll.bBusy THEN
			RETURN;
		ELSIF hSiftClient.fbCloseAll.bError THEN
			nErrId := hSiftClient.fbCloseAll.nErrId;
			eState := FAILURE;
			nErrMsg := 'Failed to call FB_CloseAll';
			RETURN;
		END_IF
		eState := CONNECT;

	CONNECT:
		bBusy := TRUE;
		bError := FALSE;
		hSiftClient.sHost := sSiftProxyHost;
		hSiftClient.nPort := nSiftProxyPort;
		hSiftClient.sApiKey := sApiKey;
		hSiftClient.sGrpcUri := sGrpcUri;
		
		IF pJsonBuffer = 0 THEN
			nErrId := GVL_SIFT.NULL_JSON_POINTER;
			eState := FAILURE;
			RETURN;
		END_IF
		hSiftClient.pJsonBuffer := pJsonBuffer;
		hSiftClient.pJbLength := pJbLength;
		
		hSiftClient.fbConnect(sRemoteHost := sSiftProxyHost, 
						      nRemotePort := nSiftProxyPort, 
							  bExecute := TRUE,
							  tTimeout := T#1S);
		
		nAttempts := nAttempts + 1;
		IF nAttempts >= 3 THEN
			nErrId := GVL_SIFT.SIFT_PROXY_FAILED_TO_START;
			nErrMsg := 'Failed to connect to sift-proxy';
			eState := FAILURE;
			RETURN;
		END_IF
		
		eState := CONNECT_WAIT;
		
	CONNECT_WAIT:
		bBusy := TRUE;
		bError := FALSE;
		hSiftClient.fbConnect(bExecute := FALSE);
		
		IF hSiftClient.fbConnect.bBusy THEN
			RETURN;
		ELSIF hSiftClient.fbConnect.bError THEN
			nErrId := hSiftClient.fbConnect.nErrId;
			eState := GET_LOCAL_AMD_NET_ID;
			RETURN;
		END_IF
		eState := AUTHENTICATE;
		
	GET_LOCAL_AMD_NET_ID:
		bBusy := TRUE;
		bError := FALSE;
		fbGetLocalAmsNetID(bExecute := TRUE);
		eState := GET_LOCAL_AMD_NET_ID_WAIT;
		
	GET_LOCAL_AMD_NET_ID_WAIT:
		bBusy := TRUE;
		bError := FALSE;
		fbGetLocalAmsNetID(bExecute := FALSE);
		
		IF fbGetLocalAmsNetID.bBusy THEN
			RETURN;
		ELSIF fbGetLocalAmsNetID.bError THEN
			nErrId := fbGetLocalAmsNetID.nErrId;
			nErrMsg := 'Failed to get local AmsNetId';
			eState := FAILURE;
			RETURN;
		END_IF
		eState := START_SIFT_PROXY;

	START_SIFT_PROXY:
		bBusy := TRUE;
		bError := FALSE;
		IF sGrpcUri = '' THEN
			nErrId := GVL_SIFT.INVALID_GRPC_URI;
			nErrMsg := 'GRPC URI not set';
			eState := FAILURE;
			RETURN;
		END_IF
		IF sApiKey = '' THEN
			nErrId := GVL_SIFT.INVALID_API_KEY;
			nErrMsg := 'API Key not set';
			eState := FAILURE;
			RETURN;
		END_IF
		IF sLogDir = '' THEN
			nErrId := GVL_SIFT.INVALID_LOG_DIR;
			nErrMsg := 'Log directory not set';
			eState := FAILURE;
			RETURN;
		END_IF
				
		fbFormat(
			sFormat := GVL_SIFT.SIFT_PROXY_CMD_ARGS, 
			arg1 := F_STRING(sLogDir),
			arg2 := F_UINT(nSiftProxyPort), 
			arg3 := F_STRING(sGrpcUri), 
			arg4 := F_STRING(sApiKey),
		);
		IF fbFormat.bError THEN
			nErrId := fbFormat.nErrId;
			nErrMsg := 'Failed to create sift-proxy command';
			eState := FAILURE;
		END_IF
		
		fbStartSiftProxy(
			NetId:=fbGetLocalAmsNetID.AddrString,
			PATHSTR:=SiftClientParameters.START_SIFT_PROXY_PATH, 
			COMNDLINE:=fbFormat.sOut,
			START := TRUE,
		);

		eState := START_SIFT_PROXY_WAIT;
				
	START_SIFT_PROXY_WAIT:
		bBusy := TRUE;
		bError := FALSE;
		fbStartSiftProxy(START := FALSE);
		
		IF fbStartSiftProxy.BUSY THEN
			RETURN;
		ELSIF fbStartSiftProxy.ERR THEN
			nErrId := fbStartSiftProxy.ERRID;
			nErrMsg := 'Failed to start sift-proxy';
			eState := FAILURE;
			RETURN;
		END_IF

		startDelay(IN:=FALSE);
		startDelay(IN:=TRUE, PT:=GVL_SIFT.SIFT_PROXY_START_DELAY);
		
		eState := START_SIFT_PROXY_DELAY;

	START_SIFT_PROXY_DELAY:
		bBusy := TRUE;
		bError := FALSE;
		
		startDelay();
		IF NOT startDelay.Q THEN
			RETURN;
		END_IF
		
		eState := CONNECT;
		
	AUTHENTICATE:
		bBusy := TRUE;
		bError := FALSE;
		fbAuth(hSiftClient:=hSiftClient, bExecute:=TRUE);
		eState := AUTHENTICATE_WAIT;
		
	AUTHENTICATE_WAIT:
		bBusy := TRUE;
		bError := FALSE;
		fbAuth(bExecute:=FALSE);
		
		IF fbAuth.bBusy THEN
			RETURN;
		ELSIF fbAuth.bError THEN
			nErrId := fbAuth.nErrId;
			nErrMsg := 'Failed to authenticate';
			eState := FAILURE;
			RETURN;
		END_IF
		eState := SUCCESS;
		
	SUCCESS:
		bBusy := FALSE;
		bError := FALSE;
		eState := IDLE;
		
	FAILURE:
		bBusy := FALSE;
		bError := TRUE;
		eState := IDLE;
		
	STOP:
		bBusy := TRUE;
		bError := FALSE;
		hSiftClient.fbCloseAll(bExecute := TRUE);
		eState := STOP_WAIT;
		
	STOP_WAIT:
		bBusy := TRUE;
		bError := FALSE;
		hSiftClient.fbCloseAll(bExecute := FALSE);
		
		IF hSiftClient.fbCloseAll.bBusy THEN
			RETURN;
		ELSIF hSiftClient.fbCloseAll.bError THEN
			nErrId := hSiftClient.fbCloseAll.nErrId;
			nErrMsg := 'Failed to call FB_CloseAll';
			eState := FAILURE;
			RETURN;
		END_IF
		eState := IDLE;
END_CASE

END_FUNCTION_BLOCK

// ---- POUs/Services/Private/FB_AuthenticateService.TcPOU
FUNCTION_BLOCK FB_AuthenticateService
VAR_INPUT
	hSiftClient : T_SiftClient;
	bExecute : BOOL;
END_VAR

VAR_OUTPUT
	bBusy : BOOL;
	bError : BOOL;
	nErrId : UDINT;
	bSuccess : BOOL;
	stSiftError : ST_SiftError;
END_VAR

VAR
END_VAR

VAR
	eState : (IDLE, SEND_MESSAGE, WAIT_FOR_RESPONSE, SUCCESS, FAILURE) := IDLE;
	fbSendSiftMessage : _FB_SendSiftMessage;
	stAuthReq : _ST_SiftMessage;
	fbJson : FB_JsonDomParser;
	sResponse : STRING(GVL_SIFT.MAX_JSON_RESPONSE_SIZE);
	jsonDoc : SJsonValue;
END_VAR

CASE eState OF
	IDLE:
		IF bExecute THEN
			eState := SEND_MESSAGE;
		END_IF
		
	SEND_MESSAGE:
		bBusy := TRUE;
		bError := FALSE;
		
		stSiftError := _F_CreateAuthenticateMessage(sApiKey:=hSiftClient.sApiKey, 
			                                        sGrpcUri:=hSiftClient.sGrpcUri, 
													pJsonBuffer := hSiftClient.pJsonBuffer,
													nLength := hSiftClient.pJbLength,
                                                    stMsg:=stAuthReq);
		IF stSiftError.bError THEN
			nErrId := stSiftError.nErrId;
			eState := FAILURE;
		END_IF
		
		fbSendSiftMessage(hSiftClient:=hSiftClient, stMsg:=stAuthReq, bExecute:=TRUE);
		eState := WAIT_FOR_RESPONSE;

	WAIT_FOR_RESPONSE:
		bBusy := TRUE;
		bError := FALSE;
		fbSendSiftMessage(bExecute:=FALSE);
		
		IF fbSendSiftMessage.bBusy THEN
			RETURN;
		ELSIF fbSendSiftMessage.bError THEN
			nErrId := fbSendSiftMessage.nErrId;
			eState := FAILURE;
			RETURN;
		END_IF

		// Verify response.
		IF fbSendSiftMessage.stResponse.nLength > GVL_SIFT.MAX_JSON_RESPONSE_SIZE THEN
			nErrId := GVL_SIFT.JSON_CAPACITY_REACHED;
			eState := FAILURE;
			RETURN;	
		END_IF
		
		IF NOT SAFE_MEMCPY(ADR(sResponse), SIZEOF(sResponse), 
			               ADR(fbSendSiftMessage.stResponse.aData), fbSendSiftMessage.stResponse.nLength) THEN
			nErrId := GVL_SIFT.MEMCPY_ERROR;
			eState := FAILURE;
		END_IF
		
		jsonDoc := fbJson.ParseDocument(sResponse);
		IF jsonDoc = 0 THEN
			eState := FAILURE;
			nErrId := GVL_SIFT.UNABLE_TO_PARSE_JSON;
		END_IF
		
		IF _F_IsSuccessfulResponse(jsonDoc) THEN
			eState := SUCCESS;
		ELSE
			IF NOT _F_SetSiftError(jsonDoc, stSiftError) THEN
				nErrId := GVL_SIFT.SIFT_PROXY_INVALID_RESPONSE;
			END_IF
			nErrId := stSiftError.nErrId;
			eState := FAILURE;
		END_IF
		
	SUCCESS:
		bBusy := FALSE;
		bError := FALSE;
		bSuccess := TRUE;
		eState := IDLE;
		
	FAILURE:
		bBusy := FALSE;
		bError := TRUE;
		eState := IDLE;
END_CASE

END_FUNCTION_BLOCK

// ---- POUs/Private/_F_CreateAuthenticateMessage.TcPOU
// Creates a Sift Proxy Protocol "authenticate" Endpoint Message.
FUNCTION _F_CreateAuthenticateMessage
VAR_INPUT
	sApiKey : STRING(255);
	sGrpcUri : STRING(255);
	stMsg : REFERENCE TO _ST_SiftMessage;
	pJsonBuffer : POINTER TO BYTE;
	nLength : UDINT;
END_VAR

VAR
	fbJson : FB_JsonSaxWriter;
	i : UDINT;
	nBytes : UDINT;
	pJsonString: POINTER TO STRING;
END_VAR

